KUKA KRL program: EPS_2_25990_SANMH01_A_20251014010954.src

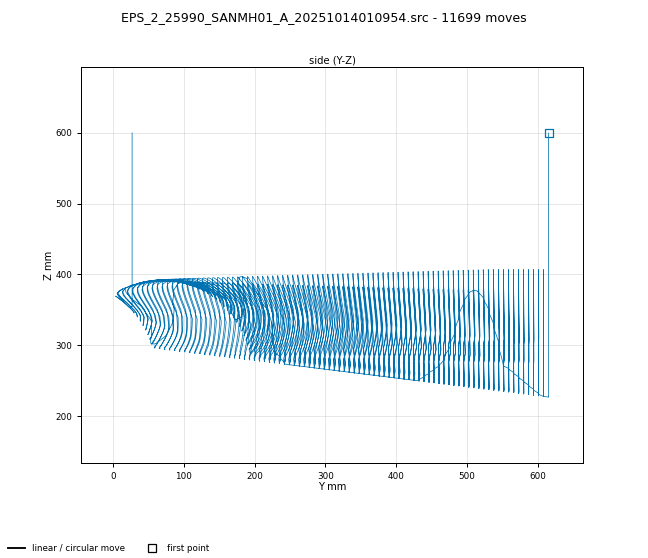
[picture p0: tool path of EPS_2_25990_SANMH01_A_20251014010954.src, 11699 of 11701 moves have a stored position in this frame; points joined in program order, loops and branches not executed]
&ACCESS RVP
&REL 4
&COMMENT QRS 19112012
&PARAM EDITMASK = *
DEF PART()
EXT BAS (BAS_COMMAND :IN,REAL :IN )
INT I
BAS (#INITMOV,0 )

;KUKA QRS Post kuka4.cps  Date:22-06-2017 !

File_ID=2882

QRS_PRE_INIT()

;Init var - Until changes are made in qrs_pre_init
Outlet_Square_prg=0
Inlet_1_Square_prg=0
Inlet_2_Square_prg=0
Inlet_3_Square_prg=0
Inlet_4_Square_prg=0
Inlet_5_Square_prg=0

Outlet_1={X 0.000, Y 531.880, Z 306.500, B 0.000, E1 0.000 }
Inlet_1={X 0.000, Y 534.050, Z 276.500, B 0.000, E1 136.000 }
Outlet_1_type=201
Inlet_1_type=201
;QRS#1=Sidecore dimensions
;QRS#2=200-8" PVC SDR 35
;QRS#3=200-8" PVC SDR 35
;QRS#4=
;QRS#5=
;QRS#6=
;QRS#7=
;QRS#8=
;QRS#9=12-08 PSX
;QRS#10=12-08 PSX
;QRS#11=
;QRS#12=
;QRS#13=
;QRS#14=
;QRS#15=
;QRS#16=1220x127x686 2,25'
;QRS#17=EPS Height
;QRS#18=407
;QRS#19=*
;QRS#20= UPDATED VERSION 22-06-2017
;QRS#21=*
Outlet_Square=0100
Inlet_1_Square=0100
Inlet_2_Square=0
Inlet_3_Square=0
Inlet_4_Square=0
Inlet_5_Square=0
Mill_Square=1
Outlet_Square_Prg=204
Inlet_1_Square_prg=204

QRS_INIT()

$ADVANCE=5

; T1
PTP {E1 173.591,E2 173.591}
PTP {X 0,Y 615.515,A -85,B 0,C 180,E1 173.591,E2 173.591,E3 0,E4 0,E5 0,E6 0}
QRS_SPEED_INIT()
LIN {X 0,Y 615.515,Z 600,A -85,B 0,C 180,E1 173.591,E2 173.591,E3 0,E4 0,E5 0,E6 0} C_VEL
LIN {X 0,Y 615.515,Z 236.872,A -85,B 0,C 180,E1 173.591,E2 173.591} C_VEL
LIN {X 0,Y 615.515,Z 228.698,A -85,B 0,C 180,E1 173.591,E2 173.591} C_VEL
LIN {X 0,Y 615.495,Z 226.698,A -85,B 0,C 180,E1 173.405,E2 173.405} C_VEL
LIN {X 0,Y 615.477,Z 226.7,A -85,B 0,C 180,E1 170.802,E2 170.802} C_VEL
LIN {X 0,Y 615.494,Z 226.697,A -85,B 0,C 180,E1 169.474,E2 169.474} C_VEL
LIN {X 0,Y 615.459,Z 228.778,A -85,B 0,C 180,E1 168.14,E2 168.14} C_VEL
LIN {X 0,Y 615.473,Z 233.515,A -85,B 0,C 180,E1 165.452,E2 165.452} C_VEL
LIN {X 0,Y 615.488,Z 238.387,A -85,B 0,C 180,E1 162.73,E2 162.73} C_VEL
LIN {X 0,Y 615.488,Z 243.54,A -85,B 0,C 180,E1 159.968,E2 159.968} C_VEL
LIN {X 0,Y 615.486,Z 248.916,A -85,B 0,C 180,E1 157.156,E2 157.156} C_VEL
LIN {X 0,Y 615.468,Z 254.224,A -85,B 0,C 180,E1 154.432,E2 154.432} C_VEL
LIN {X 0,Y 615.487,Z 259.957,A -85,B 0,C 180,E1 151.548,E2 151.548} C_VEL
LIN {X 0,Y 615.466,Z 265.253,A -85,B 0,C 180,E1 148.915,E2 148.915} C_VEL
LIN {X 0,Y 615.466,Z 270.245,A -85,B 0,C 180,E1 146.467,E2 146.467} C_VEL
LIN {X 0,Y 615.49,Z 272.215,A -85,B 0,C 180,E1 145.555,E2 145.555} C_VEL
LIN {X 0,Y 615.481,Z 285.466,A -85,B 0,C 180,E1 145.27,E2 145.27} C_VEL
LIN {X 0,Y 615.458,Z 298.826,A -85,B 0,C 180,E1 144.835,E2 144.835} C_VEL
LIN {X 0,Y 615.475,Z 310.215,A -85,B 0,C 180,E1 144.329,E2 144.329} C_VEL
LIN {X 0,Y 615.489,Z 322.006,A -85,B 0,C 180,E1 143.65,E2 143.65} C_VEL
LIN {X 0,Y 615.498,Z 332.274,A -85,B 0,C 180,E1 142.91,E2 142.91} C_VEL
LIN {X 0,Y 615.495,Z 340.609,A -85,B 0,C 180,E1 142.18,E2 142.18} C_VEL
LIN {X 0,Y 615.497,Z 348.841,A -85,B 0,C 180,E1 141.308,E2 141.308} C_VEL
LIN {X 0,Y 615.494,Z 356.847,A -85,B 0,C 180,E1 140.252,E2 140.252} C_VEL
LIN {X 0,Y 615.495,Z 363.456,A -85,B 0,C 180,E1 139.15,E2 139.15} C_VEL
LIN {X 0,Y 615.495,Z 367.798,A -85,B 0,C 180,E1 138.224,E2 138.224} C_VEL
LIN {X 0,Y 615.494,Z 371.164,A -85,B 0,C 180,E1 137.301,E2 137.301} C_VEL
LIN {X 0,Y 615.493,Z 374.47,A -85,B 0,C 180,E1 136.001,E2 136.001} C_VEL
LIN {X 0,Y 615.493,Z 375.946,A -85,B 0,C 180,E1 134.934,E2 134.934} C_VEL
LIN {X 0,Y 615.493,Z 376.384,A -85,B 0,C 180,E1 134,E2 134} C_VEL
LIN {X 0,Y 615.492,Z 375.997,A -85,B 0,C 180,E1 133.05,E2 133.05} C_VEL
LIN {X 0,Y 615.494,Z 374.759,A -85,B 0,C 180,E1 132.083,E2 132.083} C_VEL
LIN {X 0,Y 615.495,Z 372.591,A -85,B 0,C 180,E1 131.097,E2 131.097} C_VEL
LIN {X 0,Y 615.496,Z 369.385,A -85,B 0,C 180,E1 130.092,E2 130.092} C_VEL
LIN {X 0,Y 615.493,Z 364.194,A -85,B 0,C 180,E1 128.903,E2 128.903} C_VEL
LIN {X 0,Y 615.497,Z 357.942,A -85,B 0,C 180,E1 127.82,E2 127.82} C_VEL
LIN {X 0,Y 615.493,Z 350.544,A -85,B 0,C 180,E1 126.81,E2 126.81} C_VEL
LIN {X 0,Y 615.498,Z 341.718,A -85,B 0,C 180,E1 125.837,E2 125.837} C_VEL
LIN {X 0,Y 615.497,Z 332.446,A -85,B 0,C 180,E1 125.013,E2 125.013} C_VEL
LIN {X 0,Y 615.465,Z 320.994,A -85,B 0,C 180,E1 124.193,E2 124.193} C_VEL
LIN {X 0,Y 615.415,Z 310.393,A -85,B 0,C 180,E1 123.588,E2 123.588} C_VEL
LIN {X 0,Y 615.427,Z 298.003,A -85,B 0,C 180,E1 123.044,E2 123.044} C_VEL
LIN {X 0,Y 615.47,Z 285.899,A -85,B 0,C 180,E1 122.652,E2 122.652} C_VEL
LIN {X 0,Y 615.479,Z 272.071,A -85,B 0,C 180,E1 122.332,E2 122.332} C_VEL
LIN {X 0,Y 615.417,Z 266.106,A -85,B 0,C 180,E1 119.409,E2 119.409} C_VEL
LIN {X 0,Y 615.448,Z 261.314,A -85,B 0,C 180,E1 117.041,E2 117.041} C_VEL
LIN {X 0,Y 615.457,Z 255.808,A -85,B 0,C 180,E1 114.273,E2 114.273} C_VEL
LIN {X 0,Y 615.443,Z 251.613,A -85,B 0,C 180,E1 112.138,E2 112.138} C_VEL
LIN {X 0,Y 615.436,Z 247.54,A -85,B 0,C 180,E1 110.034,E2 110.034} C_VEL
LIN {X 0,Y 615.433,Z 243.584,A -85,B 0,C 180,E1 107.958,E2 107.958} C_VEL
LIN {X 0,Y 615.436,Z 239.741,A -85,B 0,C 180,E1 105.906,E2 105.906} C_VEL
LIN {X 0,Y 615.485,Z 234.819,A -85,B 0,C 180,E1 103.201,E2 103.201} C_VEL
LIN {X 0,Y 615.495,Z 230.063,A -85,B 0,C 180,E1 100.526,E2 100.526} C_VEL
LIN {X 0,Y 615.478,Z 226.7,A -85,B 0,C 180,E1 98.536,E2 98.536} C_VEL
LIN {X 0,Y 615.468,Z 226.7,A -85,B 0,C 180,E1 95.899,E2 95.899} C_VEL
LIN {X 0,Y 615.476,Z 226.698,A -85,B 0,C 180,E1 93.273,E2 93.273} C_VEL
LIN {X 0,Y 615.489,Z 226.697,A -85,B 0,C 180,E1 90.654,E2 90.654} C_VEL
LIN {X 0,Y 615.495,Z 226.7,A -85,B 0,C 180,E1 88.037,E2 88.037} C_VEL
LIN {X 0,Y 615.495,Z 226.698,A -85,B 0,C 180,E1 85.415,E2 85.415} C_VEL
LIN {X 0,Y 615.475,Z 226.699,A -85,B 0,C 180,E1 82.784,E2 82.784} C_VEL
LIN {X 0,Y 615.464,Z 226.701,A -85,B 0,C 180,E1 80.138,E2 80.138} C_VEL
LIN {X 0,Y 615.478,Z 226.699,A -85,B 0,C 180,E1 77.47,E2 77.47} C_VEL
LIN {X 0,Y 615.492,Z 226.702,A -85,B 0,C 180,E1 74.774,E2 74.774} C_VEL
LIN {X 0,Y 615.475,Z 226.699,A -85,B 0,C 180,E1 72.043,E2 72.043} C_VEL
LIN {X 0,Y 615.492,Z 226.694,A -85,B 0,C 180,E1 69.27,E2 69.27} C_VEL
LIN {X 0,Y 615.484,Z 226.702,A -85,B 0,C 180,E1 66.444,E2 66.444} C_VEL
LIN {X 0,Y 615.493,Z 226.695,A -85,B 0,C 180,E1 63.557,E2 63.557} C_VEL
LIN {X 0,Y 615.482,Z 226.7,A -85,B 0,C 180,E1 60.594,E2 60.594} C_VEL
LIN {X 0,Y 615.473,Z 226.7,A -85,B 0,C 180,E1 58.314,E2 58.314} C_VEL
LIN {X 0,Y 615.469,Z 226.7,A -85,B 0,C 180,E1 55.977,E2 55.977} C_VEL
LIN {X 0,Y 615.491,Z 226.695,A -85,B 0,C 180,E1 53.576,E2 53.576} C_VEL
LIN {X 0,Y 615.49,Z 226.699,A -85,B 0,C 180,E1 50.936,E2 50.936} C_VEL
LIN {X 0,Y 615.484,Z 226.7,A -85,B 0,C 180,E1 48.527,E2 48.527} C_VEL
LIN {X 0,Y 615.499,Z 226.698,A -85,B 0,C 180,E1 45.852,E2 45.852} C_VEL
LIN {X 0,Y 615.465,Z 226.7,A -85,B 0,C 180,E1 43.046,E2 43.046} C_VEL
LIN {X 0,Y 615.467,Z 226.7,A -85,B 0,C 180,E1 40.607,E2 40.607} C_VEL
LIN {X 0,Y 615.484,Z 226.697,A -85,B 0,C 180,E1 38.013,E2 38.013} C_VEL
LIN {X 0,Y 615.487,Z 226.696,A -85,B 0,C 180,E1 35.615,E2 35.615} C_VEL
LIN {X 0,Y 615.47,Z 226.7,A -85,B 0,C 180,E1 33.236,E2 33.236} C_VEL
LIN {X 0,Y 615.467,Z 226.7,A -85,B 0,C 180,E1 30.92,E2 30.92} C_VEL
LIN {X 0,Y 615.472,Z 226.699,A -85,B 0,C 180,E1 28.449,E2 28.449} C_VEL
LIN {X 0,Y 615.498,Z 226.7,A -85,B 0,C 180,E1 25.573,E2 25.573} C_VEL
LIN {X 0,Y 615.477,Z 226.699,A -85,B 0,C 180,E1 22.844,E2 22.844} C_VEL
LIN {X 0,Y 615.493,Z 226.694,A -85,B 0,C 180,E1 20.032,E2 20.032} C_VEL
LIN {X 0,Y 615.488,Z 226.701,A -85,B 0,C 180,E1 17.269,E2 17.269} C_VEL
LIN {X 0,Y 615.494,Z 226.697,A -85,B 0,C 180,E1 14.548,E2 14.548} C_VEL
LIN {X 0,Y 615.472,Z 226.699,A -85,B 0,C 180,E1 11.86,E2 11.86} C_VEL
LIN {X 0,Y 615.469,Z 226.7,A -85,B 0,C 180,E1 9.198,E2 9.198} C_VEL
LIN {X 0,Y 615.485,Z 226.7,A -85,B 0,C 180,E1 6.556,E2 6.556} C_VEL
LIN {X 0,Y 615.487,Z 226.702,A -85,B 0,C 180,E1 3.928,E2 3.928} C_VEL
LIN {X 0,Y 615.48,Z 226.699,A -85,B 0,C 180,E1 1.308,E2 1.308} C_VEL
LIN {X 0,Y 615.493,Z 226.694,A -85,B 0,C 180,E1 -1.309,E2 -1.309} C_VEL
LIN {X 0,Y 615.477,Z 226.698,A -85,B 0,C 180,E1 -3.929,E2 -3.929} C_VEL
LIN {X 0,Y 615.477,Z 226.7,A -85,B 0,C 180,E1 -6.578,E2 -6.578} C_VEL
LIN {X 0,Y 615.496,Z 226.7,A -85,B 0,C 180,E1 -9.199,E2 -9.199} C_VEL
LIN {X 0,Y 615.479,Z 226.7,A -85,B 0,C 180,E1 -11.862,E2 -11.862} C_VEL
LIN {X 0,Y 615.467,Z 226.7,A -85,B 0,C 180,E1 -14.55,E2 -14.55} C_VEL
LIN {X 0,Y 615.496,Z 226.695,A -85,B 0,C 180,E1 -17.271,E2 -17.271} C_VEL
LIN {X 0,Y 615.489,Z 226.702,A -85,B 0,C 180,E1 -20.033,E2 -20.033} C_VEL
LIN {X 0,Y 615.489,Z 226.696,A -85,B 0,C 180,E1 -22.845,E2 -22.845} C_VEL
LIN {X 0,Y 615.477,Z 226.699,A -85,B 0,C 180,E1 -25.717,E2 -25.717} C_VEL
LIN {X 0,Y 615.499,Z 226.7,A -85,B 0,C 180,E1 -28.454,E2 -28.454} C_VEL
LIN {X 0,Y 615.486,Z 226.698,A -85,B 0,C 180,E1 -31.087,E2 -31.087} C_VEL
LIN {X 0,Y 615.475,Z 226.7,A -85,B 0,C 180,E1 -33.534,E2 -33.534} C_VEL
LIN {X 0,Y 615.481,Z 226.7,A -85,B 0,C 180,E1 -35.834,E2 -35.834} C_VEL
LIN {X 0,Y 615.488,Z 226.702,A -85,B 0,C 180,E1 -38.069,E2 -38.069} C_VEL
LIN {X 0,Y 615.486,Z 226.696,A -85,B 0,C 180,E1 -41.095,E2 -41.095} C_VEL
LIN {X 0,Y 615.493,Z 226.699,A -85,B 0,C 180,E1 -44.15,E2 -44.15} C_VEL
LIN {X 0,Y 615.485,Z 226.696,A -85,B 0,C 180,E1 -46.953,E2 -46.953} C_VEL
LIN {X 0,Y 615.467,Z 226.7,A -85,B 0,C 180,E1 -49.393,E2 -49.393} C_VEL
LIN {X 0,Y 615.469,Z 226.7,A -85,B 0,C 180,E1 -51.991,E2 -51.991} C_VEL
LIN {X 0,Y 615.491,Z 226.813,A -85,B 0,C 180,E1 -54.586,E2 -54.586} C_VEL
LIN {X 0,Y 615.479,Z 233.99,A -85,B 0,C 180,E1 -57.154,E2 -57.154} C_VEL
LIN {X 0,Y 615.46,Z 241.78,A -85,B 0,C 180,E1 -59.839,E2 -59.839} C_VEL
LIN {X 0,Y 615.492,Z 249.544,A -85,B 0,C 180,E1 -62.455,E2 -62.455} C_VEL
LIN {X 0,Y 615.442,Z 257.313,A -85,B 0,C 180,E1 -65.007,E2 -65.007} C_VEL
LIN {X 0,Y 615.47,Z 265.535,A -85,B 0,C 180,E1 -67.659,E2 -67.659} C_VEL
LIN {X 0,Y 615.487,Z 273.927,A -85,B 0,C 180,E1 -70.315,E2 -70.315} C_VEL
LIN {X 0,Y 615.484,Z 282.785,A -85,B 0,C 180,E1 -73.072,E2 -73.072} C_VEL
LIN {X 0,Y 615.469,Z 291.547,A -85,B 0,C 180,E1 -75.76,E2 -75.76} C_VEL
LIN {X 0,Y 615.496,Z 300.138,A -85,B 0,C 180,E1 -78.369,E2 -78.369} C_VEL
LIN {X 0,Y 615.497,Z 313.826,A -85,B 0,C 180,E1 -78.64,E2 -78.64} C_VEL
LIN {X 0,Y 615.455,Z 326.951,A -85,B 0,C 180,E1 -79.05,E2 -79.05} C_VEL
LIN {X 0,Y 615.447,Z 338.775,A -85,B 0,C 180,E1 -79.556,E2 -79.556} C_VEL
LIN {X 0,Y 615.497,Z 349.388,A -85,B 0,C 180,E1 -80.138,E2 -80.138} C_VEL
LIN {X 0,Y 615.498,Z 360.233,A -85,B 0,C 180,E1 -80.884,E2 -80.884} C_VEL
LIN {X 0,Y 615.497,Z 370.812,A -85,B 0,C 180,E1 -81.794,E2 -81.794} C_VEL
LIN {X 0,Y 615.498,Z 378.606,A -85,B 0,C 180,E1 -82.62,E2 -82.62} C_VEL
LIN {X 0,Y 615.496,Z 386.203,A -85,B 0,C 180,E1 -83.608,E2 -83.608} C_VEL
LIN {X 0,Y 615.498,Z 393.204,A -85,B 0,C 180,E1 -84.759,E2 -84.759} C_VEL
LIN {X 0,Y 615.494,Z 397.851,A -85,B 0,C 180,E1 -85.744,E2 -85.744} C_VEL
LIN {X 0,Y 615.494,Z 401.399,A -85,B 0,C 180,E1 -86.727,E2 -86.727} C_VEL
LIN {X 0,Y 615.497,Z 403.233,A -85,B 0,C 180,E1 -87.382,E2 -87.382} C_VEL
LIN {X 0,Y 615.5,Z 404.607,A -85,B 0,C 180,E1 -88.037,E2 -88.037} C_VEL
LIN {X 0,Y 615.496,Z 406.173,A -85,B 0,C 180,E1 -89.346,E2 -89.346} C_VEL
LIN {X 0,Y 615.494,Z 406.389,A -85,B 0,C 180,E1 -90,E2 -90} C_VEL
LIN {X 0,Y 615.495,Z 405.58,A -85,B 0,C 180,E1 -91.308,E2 -91.308} C_VEL
LIN {X 0,Y 615.5,Z 404.608,A -85,B 0,C 180,E1 -91.963,E2 -91.963} C_VEL
LIN {X 0,Y 615.497,Z 403.233,A -85,B 0,C 180,E1 -92.618,E2 -92.618} C_VEL
LIN {X 0,Y 615.496,Z 400.35,A -85,B 0,C 180,E1 -93.6,E2 -93.6} C_VEL
LIN {X 0,Y 615.498,Z 396.442,A -85,B 0,C 180,E1 -94.584,E2 -94.584} C_VEL
LIN {X 0,Y 615.499,Z 391.406,A -85,B 0,C 180,E1 -95.569,E2 -95.569} C_VEL
LIN {X 0,Y 615.497,Z 384.871,A -85,B 0,C 180,E1 -96.583,E2 -96.583} C_VEL
LIN {X 0,Y 615.497,Z 377.135,A -85,B 0,C 180,E1 -97.545,E2 -97.545} C_VEL
LIN {X 0,Y 615.498,Z 369.048,A -85,B 0,C 180,E1 -98.371,E2 -98.371} C_VEL
LIN {X 0,Y 615.499,Z 359.171,A -85,B 0,C 180,E1 -99.198,E2 -99.198} C_VEL
LIN {X 0,Y 615.486,Z 347.987,A -85,B 0,C 180,E1 -99.945,E2 -99.945} C_VEL
LIN {X 0,Y 615.445,Z 337.036,A -85,B 0,C 180,E1 -100.527,E2 -100.527} C_VEL
LIN {X 0,Y 615.461,Z 324.766,A -85,B 0,C 180,E1 -101.031,E2 -101.031} C_VEL
LIN {X 0,Y 615.498,Z 312.077,A -85,B 0,C 180,E1 -101.401,E2 -101.401} C_VEL
LIN {X 0,Y 615.496,Z 300.139,A -85,B 0,C 180,E1 -101.631,E2 -101.631} C_VEL
LIN {X 0,Y 615.469,Z 291.548,A -85,B 0,C 180,E1 -104.24,E2 -104.24} C_VEL
LIN {X 0,Y 615.484,Z 282.786,A -85,B 0,C 180,E1 -106.928,E2 -106.928} C_VEL
LIN {X 0,Y 615.487,Z 273.928,A -85,B 0,C 180,E1 -109.684,E2 -109.684} C_VEL
LIN {X 0,Y 615.474,Z 265.532,A -85,B 0,C 180,E1 -112.342,E2 -112.342} C_VEL
LIN {X 0,Y 615.442,Z 257.313,A -85,B 0,C 180,E1 -114.993,E2 -114.993} C_VEL
LIN {X 0,Y 615.492,Z 249.545,A -85,B 0,C 180,E1 -117.545,E2 -117.545} C_VEL
LIN {X 0,Y 615.46,Z 241.779,A -85,B 0,C 180,E1 -120.161,E2 -120.161} C_VEL
LIN {X 0,Y 615.478,Z 233.974,A -85,B 0,C 180,E1 -122.846,E2 -122.846} C_VEL
LIN {X 0,Y 615.492,Z 226.697,A -85,B 0,C 180,E1 -125.514,E2 -125.514} C_VEL
LIN {X 0,Y 615.488,Z 226.699,A -85,B 0,C 180,E1 -128.068,E2 -128.068} C_VEL
LIN {X 0,Y 615.48,Z 226.7,A -85,B 0,C 180,E1 -130.606,E2 -130.606} C_VEL
LIN {X 0,Y 615.497,Z 226.698,A -85,B 0,C 180,E1 -133.243,E2 -133.243} C_VEL
LIN {X 0,Y 615.476,Z 226.7,A -85,B 0,C 180,E1 -136.002,E2 -136.002} C_VEL
LIN {X 0,Y 615.49,Z 226.697,A -85,B 0,C 180,E1 -138.904,E2 -138.904} C_VEL
LIN {X 0,Y 615.495,Z 226.696,A -85,B 0,C 180,E1 -141.096,E2 -141.096} C_VEL
LIN {X 0,Y 615.491,Z 226.701,A -85,B 0,C 180,E1 -143.575,E2 -143.575} C_VEL
LIN {X 0,Y 615.481,Z 226.7,A -85,B 0,C 180,E1 -145.977,E2 -145.977} C_VEL
LIN {X 0,Y 615.473,Z 226.701,A -85,B 0,C 180,E1 -148.313,E2 -148.313} C_VEL
LIN {X 0,Y 615.478,Z 226.701,A -85,B 0,C 180,E1 -150.593,E2 -150.593} C_VEL
LIN {X 0,Y 615.498,Z 226.699,A -85,B 0,C 180,E1 -152.951,E2 -152.951} C_VEL
LIN {X 0,Y 615.494,Z 226.701,A -85,B 0,C 180,E1 -155.988,E2 -155.988} C_VEL
LIN {X 0,Y 615.484,Z 226.698,A -85,B 0,C 180,E1 -158.567,E2 -158.567} C_VEL
LIN {X 0,Y 615.48,Z 226.7,A -85,B 0,C 180,E1 -161.394,E2 -161.394} C_VEL
LIN {X 0,Y 615.486,Z 226.701,A -85,B 0,C 180,E1 -164.094,E2 -164.094} C_VEL
LIN {X 0,Y 615.497,Z 226.695,A -85,B 0,C 180,E1 -166.798,E2 -166.798} C_VEL
LIN {X 0,Y 615.484,Z 226.701,A -85,B 0,C 180,E1 -169.472,E2 -169.472} C_VEL
LIN {X 0,Y 615.481,Z 226.7,A -85,B 0,C 180,E1 -172.124,E2 -172.124} C_VEL
LIN {X 0,Y 615.489,Z 226.698,A -85,B 0,C 180,E1 -174.758,E2 -174.758} C_VEL
LIN {X 0,Y 615.489,Z 226.7,A -85,B 0,C 180,E1 -177.381,E2 -177.381} C_VEL
LIN {X 0,Y 615.478,Z 226.7,A -85,B 0,C 180,E1 -179.999,E2 -179.999} C_VEL
LIN {X 0,Y 615.495,Z 226.7,A -85,B 0,C 180,E1 -182.617,E2 -182.617} C_VEL
LIN {X 0,Y 615.474,Z 226.7,A -85,B 0,C 180,E1 -185.24,E2 -185.24} C_VEL
LIN {X 0,Y 615.495,Z 226.698,A -85,B 0,C 180,E1 -186.595,E2 -186.595} C_VEL
LIN {X 0,Y 614.805,Z 226.845,A -85,B 0,C 180,E1 -187.141,E2 -187.141} C_VEL
LIN {X 0,Y 611.958,Z 227.26,A -85,B 0,C 180,E1 -188.027,E2 -188.027} C_VEL
LIN {X 0,Y 609.568,Z 227.568,A -85,B 0,C 180,E1 -188.739,E2 -188.739} C_VEL
LIN {X 0,Y 608.541,Z 227.685,A -85,B 0,C 180,E1 -189.289,E2 -189.289} C_VEL
LIN {X 0,Y 608.457,Z 227.694,A -85,B 0,C 180,E1 -189.475,E2 -189.475} C_VEL
LIN {X 0,Y 608.443,Z 227.698,A -85,B 0,C 180,E1 -190.649,E2 -190.649} C_VEL
LIN {X 0,Y 608.431,Z 232.361,A -85,B 0,C 180,E1 -193.356,E2 -193.356} C_VEL
LIN {X 0,Y 608.445,Z 237.188,A -85,B 0,C 180,E1 -196.093,E2 -196.093} C_VEL
LIN {X 0,Y 608.448,Z 242.225,A -85,B 0,C 180,E1 -198.869,E2 -198.869} C_VEL
LIN {X 0,Y 608.438,Z 247.537,A -85,B 0,C 180,E1 -201.692,E2 -201.692} C_VEL
LIN {X 0,Y 608.424,Z 253.079,A -85,B 0,C 180,E1 -204.571,E2 -204.571} C_VEL
LIN {X 0,Y 608.415,Z 258.231,A -85,B 0,C 180,E1 -207.198,E2 -207.198} C_VEL
LIN {X 0,Y 608.448,Z 263.754,A -85,B 0,C 180,E1 -209.97,E2 -209.97} C_VEL
LIN {X 0,Y 608.414,Z 269.639,A -85,B 0,C 180,E1 -212.881,E2 -212.881} C_VEL
LIN {X 0,Y 608.442,Z 272.542,A -85,B 0,C 180,E1 -214.305,E2 -214.305} C_VEL
LIN {X 0,Y 608.52,Z 287.737,A -85,B 0,C 180,E1 -214.659,E2 -214.659} C_VEL
LIN {X 0,Y 608.501,Z 299.429,A -85,B 0,C 180,E1 -215.057,E2 -215.057} C_VEL
LIN {X 0,Y 608.478,Z 310.914,A -85,B 0,C 180,E1 -215.579,E2 -215.579} C_VEL
LIN {X 0,Y 608.496,Z 323.052,A -85,B 0,C 180,E1 -216.292,E2 -216.292} C_VEL
LIN {X 0,Y 608.485,Z 333.177,A -85,B 0,C 180,E1 -217.037,E2 -217.037} C_VEL
LIN {X 0,Y 608.468,Z 342.371,A -85,B 0,C 180,E1 -217.868,E2 -217.868} C_VEL
LIN {X 0,Y 608.444,Z 350.491,A -85,B 0,C 180,E1 -218.765,E2 -218.765} C_VEL
LIN {X 0,Y 608.437,Z 357.135,A -85,B 0,C 180,E1 -219.655,E2 -219.655} C_VEL
LIN {X 0,Y 608.435,Z 363.654,A -85,B 0,C 180,E1 -220.738,E2 -220.738} C_VEL
LIN {X 0,Y 608.449,Z 368.088,A -85,B 0,C 180,E1 -221.673,E2 -221.673} C_VEL
LIN {X 0,Y 608.438,Z 370.653,A -85,B 0,C 180,E1 -222.333,E2 -222.333} C_VEL
LIN {X 0,Y 608.431,Z 373.569,A -85,B 0,C 180,E1 -223.306,E2 -223.306} C_VEL
LIN {X 0,Y 608.418,Z 375.537,A -85,B 0,C 180,E1 -224.261,E2 -224.261} C_VEL
LIN {X 0,Y 608.415,Z 376.656,A -85,B 0,C 180,E1 -225.202,E2 -225.202} C_VEL
LIN {X 0,Y 608.426,Z 376.987,A -85,B 0,C 180,E1 -226.128,E2 -226.128} C_VEL
LIN {X 0,Y 608.431,Z 376.549,A -85,B 0,C 180,E1 -227.039,E2 -227.039} C_VEL
LIN {X 0,Y 608.422,Z 375.358,A -85,B 0,C 180,E1 -227.936,E2 -227.936} C_VEL
LIN {X 0,Y 608.431,Z 373.465,A -85,B 0,C 180,E1 -228.823,E2 -228.823} C_VEL
LIN {X 0,Y 608.438,Z 370.866,A -85,B 0,C 180,E1 -229.697,E2 -229.697} C_VEL
LIN {X 0,Y 608.45,Z 366.862,A -85,B 0,C 180,E1 -230.703,E2 -230.703} C_VEL
LIN {X 0,Y 608.434,Z 361.387,A -85,B 0,C 180,E1 -231.762,E2 -231.762} C_VEL
LIN {X 0,Y 608.443,Z 354.246,A -85,B 0,C 180,E1 -232.843,E2 -232.843} C_VEL
LIN {X 0,Y 608.459,Z 347.242,A -85,B 0,C 180,E1 -233.705,E2 -233.705} C_VEL
LIN {X 0,Y 608.476,Z 338.162,A -85,B 0,C 180,E1 -234.624,E2 -234.624} C_VEL
LIN {X 0,Y 608.477,Z 328.441,A -85,B 0,C 180,E1 -235.421,E2 -235.421} C_VEL
LIN {X 0,Y 608.437,Z 316.606,A -85,B 0,C 180,E1 -236.2,E2 -236.2} C_VEL
LIN {X 0,Y 608.429,Z 305.532,A -85,B 0,C 180,E1 -236.774,E2 -236.774} C_VEL
LIN {X 0,Y 608.488,Z 294.204,A -85,B 0,C 180,E1 -237.228,E2 -237.228} C_VEL
LIN {X 0,Y 608.533,Z 281.365,A -85,B 0,C 180,E1 -237.597,E2 -237.597} C_VEL
LIN {X 0,Y 608.398,Z 272.531,A -85,B 0,C 180,E1 -237.792,E2 -237.792} C_VEL
LIN {X 0,Y 608.373,Z 267.597,A -85,B 0,C 180,E1 -240.216,E2 -240.216} C_VEL
LIN {X 0,Y 608.387,Z 262.38,A -85,B 0,C 180,E1 -242.807,E2 -242.807} C_VEL
LIN {X 0,Y 608.397,Z 257.176,A -85,B 0,C 180,E1 -245.427,E2 -245.427} C_VEL
LIN {X 0,Y 608.418,Z 252.935,A -85,B 0,C 180,E1 -247.593,E2 -247.593} C_VEL
LIN {X 0,Y 608.399,Z 248.827,A -85,B 0,C 180,E1 -249.724,E2 -249.724} C_VEL
LIN {X 0,Y 608.42,Z 243.53,A -85,B 0,C 180,E1 -252.523,E2 -252.523} C_VEL
LIN {X 0,Y 608.433,Z 238.464,A -85,B 0,C 180,E1 -255.279,E2 -255.279} C_VEL
LIN {X 0,Y 608.461,Z 233.611,A -85,B 0,C 180,E1 -258.001,E2 -258.001} C_VEL
LIN {X 0,Y 608.42,Z 228.894,A -85,B 0,C 180,E1 -260.694,E2 -260.694} C_VEL
LIN {X 0,Y 608.446,Z 227.736,A -85,B 0,C 180,E1 -261.364,E2 -261.364} C_VEL
LIN {X 0,Y 608.445,Z 227.696,A -85,B 0,C 180,E1 -264.033,E2 -264.033} C_VEL
LIN {X 0,Y 608.469,Z 227.692,A -85,B 0,C 180,E1 -266.689,E2 -266.689} C_VEL
LIN {X 0,Y 608.482,Z 227.692,A -85,B 0,C 180,E1 -269.338,E2 -269.338} C_VEL
LIN {X 0,Y 608.464,Z 227.697,A -85,B 0,C 180,E1 -271.986,E2 -271.986} C_VEL
LIN {X 0,Y 608.462,Z 227.695,A -85,B 0,C 180,E1 -274.638,E2 -274.638} C_VEL
LIN {X 0,Y 608.455,Z 227.694,A -85,B 0,C 180,E1 -277.299,E2 -277.299} C_VEL
LIN {X 0,Y 608.44,Z 227.696,A -85,B 0,C 180,E1 -279.977,E2 -279.977} C_VEL
LIN {X 0,Y 608.466,Z 227.695,A -85,B 0,C 180,E1 -282.677,E2 -282.677} C_VEL
LIN {X 0,Y 608.469,Z 227.694,A -85,B 0,C 180,E1 -285.406,E2 -285.406} C_VEL
LIN {X 0,Y 608.442,Z 227.696,A -85,B 0,C 180,E1 -288.172,E2 -288.172} C_VEL
LIN {X 0,Y 608.455,Z 227.696,A -85,B 0,C 180,E1 -290.981,E2 -290.981} C_VEL
LIN {X 0,Y 608.447,Z 227.695,A -85,B 0,C 180,E1 -293.124,E2 -293.124} C_VEL
LIN {X 0,Y 608.455,Z 227.695,A -85,B 0,C 180,E1 -295.72,E2 -295.72} C_VEL
LIN {X 0,Y 608.452,Z 227.697,A -85,B 0,C 180,E1 -298.266,E2 -298.266} C_VEL
LIN {X 0,Y 608.47,Z 227.693,A -85,B 0,C 180,E1 -300.544,E2 -300.544} C_VEL
LIN {X 0,Y 608.458,Z 227.694,A -85,B 0,C 180,E1 -302.879,E2 -302.879} C_VEL
LIN {X 0,Y 608.441,Z 227.696,A -85,B 0,C 180,E1 -305.277,E2 -305.277} C_VEL
LIN {X 0,Y 608.469,Z 227.694,A -85,B 0,C 180,E1 -308.242,E2 -308.242} C_VEL
LIN {X 0,Y 608.47,Z 227.695,A -85,B 0,C 180,E1 -310.333,E2 -310.333} C_VEL
LIN {X 0,Y 608.445,Z 227.698,A -85,B 0,C 180,E1 -312.96,E2 -312.96} C_VEL
LIN {X 0,Y 608.447,Z 227.695,A -85,B 0,C 180,E1 -315.736,E2 -315.736} C_VEL
LIN {X 0,Y 608.463,Z 227.695,A -85,B 0,C 180,E1 -318.657,E2 -318.657} C_VEL
LIN {X 0,Y 608.466,Z 227.695,A -85,B 0,C 180,E1 -321.413,E2 -321.413} C_VEL
LIN {X 0,Y 608.472,Z 227.693,A -85,B 0,C 180,E1 -323.95,E2 -323.95} C_VEL
LIN {X 0,Y 608.454,Z 227.695,A -85,B 0,C 180,E1 -326.33,E2 -326.33} C_VEL
LIN {X 0,Y 608.465,Z 227.694,A -85,B 0,C 180,E1 -328.728,E2 -328.728} C_VEL
LIN {X 0,Y 608.459,Z 227.694,A -85,B 0,C 180,E1 -331.381,E2 -331.381} C_VEL
LIN {X 0,Y 608.477,Z 227.694,A -85,B 0,C 180,E1 -334.276,E2 -334.276} C_VEL
LIN {X 0,Y 608.443,Z 227.699,A -85,B 0,C 180,E1 -336.877,E2 -336.877} C_VEL
LIN {X 0,Y 608.466,Z 227.693,A -85,B 0,C 180,E1 -339.727,E2 -339.727} C_VEL
LIN {X 0,Y 608.451,Z 227.696,A -85,B 0,C 180,E1 -342.524,E2 -342.524} C_VEL
LIN {X 0,Y 608.474,Z 227.695,A -85,B 0,C 180,E1 -345.28,E2 -345.28} C_VEL
LIN {X 0,Y 608.449,Z 227.695,A -85,B 0,C 180,E1 -348.001,E2 -348.001} C_VEL
LIN {X 0,Y 608.457,Z 227.694,A -85,B 0,C 180,E1 -350.695,E2 -350.695} C_VEL
LIN {X 0,Y 608.468,Z 227.694,A -85,B 0,C 180,E1 -353.368,E2 -353.368} C_VEL
LIN {X 0,Y 608.456,Z 227.698,A -85,B 0,C 180,E1 -356.027,E2 -356.027} C_VEL
LIN {X 0,Y 608.463,Z 227.694,A -85,B 0,C 180,E1 -358.677,E2 -358.677} C_VEL
LIN {X 0,Y 608.475,Z 227.692,A -85,B 0,C 180,E1 -361.324,E2 -361.324} C_VEL
LIN {X 0,Y 608.447,Z 227.695,A -85,B 0,C 180,E1 -363.975,E2 -363.975} C_VEL
LIN {X 0,Y 608.47,Z 227.694,A -85,B 0,C 180,E1 -366.633,E2 -366.633} C_VEL
LIN {X 0,Y 608.475,Z 227.695,A -85,B 0,C 180,E1 -369.306,E2 -369.306} C_VEL
LIN {X 0,Y 608.454,Z 227.695,A -85,B 0,C 180,E1 -372.001,E2 -372.001} C_VEL
LIN {X 0,Y 608.463,Z 227.693,A -85,B 0,C 180,E1 -374.721,E2 -374.721} C_VEL
LIN {X 0,Y 608.455,Z 227.696,A -85,B 0,C 180,E1 -377.477,E2 -377.477} C_VEL
LIN {X 0,Y 608.457,Z 227.695,A -85,B 0,C 180,E1 -380.275,E2 -380.275} C_VEL
LIN {X 0,Y 608.453,Z 227.694,A -85,B 0,C 180,E1 -383.125,E2 -383.125} C_VEL
LIN {X 0,Y 608.436,Z 227.7,A -85,B 0,C 180,E1 -386.037,E2 -386.037} C_VEL
LIN {X 0,Y 608.48,Z 227.693,A -85,B 0,C 180,E1 -388.623,E2 -388.623} C_VEL
LIN {X 0,Y 608.473,Z 227.692,A -85,B 0,C 180,E1 -391.317,E2 -391.317} C_VEL
LIN {X 0,Y 608.441,Z 227.696,A -85,B 0,C 180,E1 -393.732,E2 -393.732} C_VEL
LIN {X 0,Y 608.441,Z 227.696,A -85,B 0,C 180,E1 -396.093,E2 -396.093} C_VEL
LIN {X 0,Y 608.474,Z 227.692,A -85,B 0,C 180,E1 -398.588,E2 -398.588} C_VEL
LIN {X 0,Y 608.464,Z 227.694,A -85,B 0,C 180,E1 -401.343,E2 -401.343} C_VEL
LIN {X 0,Y 608.462,Z 227.695,A -85,B 0,C 180,E1 -404.265,E2 -404.265} C_VEL
LIN {X 0,Y 608.453,Z 227.694,A -85,B 0,C 180,E1 -407.041,E2 -407.041} C_VEL
LIN {X 0,Y 608.452,Z 227.695,A -85,B 0,C 180,E1 -409.697,E2 -409.697} C_VEL
LIN {X 0,Y 608.459,Z 227.696,A -85,B 0,C 180,E1 -412.254,E2 -412.254} C_VEL
LIN {X 0,Y 608.479,Z 227.814,A -85,B 0,C 180,E1 -414.472,E2 -414.472} C_VEL
LIN {X 0,Y 608.489,Z 235.135,A -85,B 0,C 180,E1 -417.123,E2 -417.123} C_VEL
LIN {X 0,Y 608.475,Z 241.816,A -85,B 0,C 180,E1 -419.456,E2 -419.456} C_VEL
LIN {X 0,Y 608.439,Z 249.64,A -85,B 0,C 180,E1 -422.108,E2 -422.108} C_VEL
LIN {X 0,Y 608.437,Z 257.432,A -85,B 0,C 180,E1 -424.699,E2 -424.699} C_VEL
LIN {X 0,Y 608.429,Z 265.224,A -85,B 0,C 180,E1 -427.235,E2 -427.235} C_VEL
LIN {X 0,Y 608.456,Z 274.127,A -85,B 0,C 180,E1 -430.078,E2 -430.078} C_VEL
LIN {X 0,Y 608.442,Z 283.031,A -85,B 0,C 180,E1 -432.87,E2 -432.87} C_VEL
LIN {X 0,Y 608.441,Z 290.823,A -85,B 0,C 180,E1 -435.279,E2 -435.279} C_VEL
LIN {X 0,Y 608.453,Z 300.283,A -85,B 0,C 180,E1 -438.169,E2 -438.169} C_VEL
LIN {X 0,Y 608.438,Z 300.492,A -85,B 0,C 180,E1 -438.232,E2 -438.232} C_VEL
LIN {X 0,Y 608.545,Z 314.701,A -85,B 0,C 180,E1 -438.53,E2 -438.53} C_VEL
LIN {X 0,Y 608.497,Z 327.786,A -85,B 0,C 180,E1 -438.95,E2 -438.95} C_VEL
LIN {X 0,Y 608.474,Z 338.924,A -85,B 0,C 180,E1 -439.435,E2 -439.435} C_VEL
LIN {X 0,Y 608.486,Z 349.58,A -85,B 0,C 180,E1 -440.023,E2 -440.023} C_VEL
LIN {X 0,Y 608.483,Z 360.475,A -85,B 0,C 180,E1 -440.778,E2 -440.778} C_VEL
LIN {X 0,Y 608.475,Z 371.112,A -85,B 0,C 180,E1 -441.699,E2 -441.699} C_VEL
LIN {X 0,Y 608.471,Z 378.961,A -85,B 0,C 180,E1 -442.534,E2 -442.534} C_VEL
LIN {X 0,Y 608.461,Z 386.287,A -85,B 0,C 180,E1 -443.485,E2 -443.485} C_VEL
LIN {X 0,Y 608.451,Z 391.866,A -85,B 0,C 180,E1 -444.366,E2 -444.366} C_VEL
LIN {X 0,Y 608.432,Z 396.95,A -85,B 0,C 180,E1 -445.362,E2 -445.362} C_VEL
LIN {X 0,Y 608.449,Z 400.896,A -85,B 0,C 180,E1 -446.358,E2 -446.358} C_VEL
LIN {X 0,Y 608.425,Z 403.809,A -85,B 0,C 180,E1 -447.352,E2 -447.352} C_VEL
LIN {X 0,Y 608.445,Z 405.201,A -85,B 0,C 180,E1 -448.014,E2 -448.014} C_VEL
LIN {X 0,Y 608.438,Z 406.783,A -85,B 0,C 180,E1 -449.338,E2 -449.338} C_VEL
LIN {X 0,Y 608.434,Z 407,A -85,B 0,C 180,E1 -450,E2 -450} C_VEL
LIN {X 0,Y 608.448,Z 406.184,A -85,B 0,C 180,E1 -451.324,E2 -451.324} C_VEL
LIN {X 0,Y 608.445,Z 405.202,A -85,B 0,C 180,E1 -451.986,E2 -451.986} C_VEL
LIN {X 0,Y 608.425,Z 403.81,A -85,B 0,C 180,E1 -452.648,E2 -452.648} C_VEL
LIN {X 0,Y 608.449,Z 400.897,A -85,B 0,C 180,E1 -453.642,E2 -453.642} C_VEL
LIN {X 0,Y 608.432,Z 396.951,A -85,B 0,C 180,E1 -454.638,E2 -454.638} C_VEL
LIN {X 0,Y 608.438,Z 390.878,A -85,B 0,C 180,E1 -455.801,E2 -455.801} C_VEL
LIN {X 0,Y 608.462,Z 384.237,A -85,B 0,C 180,E1 -456.799,E2 -456.799} C_VEL
LIN {X 0,Y 608.456,Z 375.991,A -85,B 0,C 180,E1 -457.8,E2 -457.8} C_VEL
LIN {X 0,Y 608.472,Z 367.539,A -85,B 0,C 180,E1 -458.636,E2 -458.636} C_VEL
LIN {X 0,Y 608.481,Z 357.095,A -85,B 0,C 180,E1 -459.473,E2 -459.473} C_VEL
LIN {X 0,Y 608.494,Z 346.761,A -85,B 0,C 180,E1 -460.144,E2 -460.144} C_VEL
LIN {X 0,Y 608.469,Z 335.846,A -85,B 0,C 180,E1 -460.714,E2 -460.714} C_VEL
LIN {X 0,Y 608.493,Z 324.086,A -85,B 0,C 180,E1 -461.186,E2 -461.186} C_VEL
LIN {X 0,Y 608.549,Z 311.281,A -85,B 0,C 180,E1 -461.554,E2 -461.554} C_VEL
LIN {X 0,Y 608.438,Z 300.493,A -85,B 0,C 180,E1 -461.767,E2 -461.767} C_VEL
LIN {X 0,Y 608.415,Z 291.936,A -85,B 0,C 180,E1 -464.38,E2 -464.38} C_VEL
LIN {X 0,Y 608.451,Z 284.145,A -85,B 0,C 180,E1 -466.784,E2 -466.784} C_VEL
LIN {X 0,Y 608.457,Z 275.241,A -85,B 0,C 180,E1 -469.57,E2 -469.57} C_VEL
LIN {X 0,Y 608.445,Z 266.13,A -85,B 0,C 180,E1 -472.472,E2 -472.472} C_VEL
LIN {X 0,Y 608.431,Z 258.545,A -85,B 0,C 180,E1 -474.936,E2 -474.936} C_VEL
LIN {X 0,Y 608.468,Z 250.754,A -85,B 0,C 180,E1 -477.516,E2 -477.516} C_VEL
LIN {X 0,Y 608.47,Z 243.471,A -85,B 0,C 180,E1 -479.971,E2 -479.971} C_VEL
LIN {X 0,Y 608.486,Z 236.091,A -85,B 0,C 180,E1 -482.525,E2 -482.525} C_VEL
LIN {X 0,Y 608.514,Z 227.958,A -85,B 0,C 180,E1 -485.475,E2 -485.475} C_VEL
LIN {X 0,Y 608.479,Z 227.693,A -85,B 0,C 180,E1 -485.681,E2 -485.681} C_VEL
LIN {X 0,Y 608.467,Z 227.696,A -85,B 0,C 180,E1 -488.24,E2 -488.24} C_VEL
LIN {X 0,Y 608.461,Z 227.697,A -85,B 0,C 180,E1 -491.342,E2 -491.342} C_VEL
LIN {X 0,Y 608.464,Z 227.694,A -85,B 0,C 180,E1 -493.869,E2 -493.869} C_VEL
LIN {X 0,Y 608.475,Z 227.694,A -85,B 0,C 180,E1 -496.689,E2 -496.689} C_VEL
LIN {X 0,Y 608.448,Z 227.698,A -85,B 0,C 180,E1 -499.67,E2 -499.67} C_VEL
LIN {X 0,Y 608.465,Z 227.694,A -85,B 0,C 180,E1 -502.253,E2 -502.253} C_VEL
LIN {X 0,Y 608.483,Z 227.692,A -85,B 0,C 180,E1 -505.088,E2 -505.088} C_VEL
LIN {X 0,Y 608.467,Z 227.695,A -85,B 0,C 180,E1 -507.905,E2 -507.905} C_VEL
LIN {X 0,Y 608.46,Z 227.695,A -85,B 0,C 180,E1 -510.219,E2 -510.219} C_VEL
LIN {X 0,Y 608.483,Z 227.694,A -85,B 0,C 180,E1 -512.79,E2 -512.79} C_VEL
LIN {X 0,Y 608.482,Z 227.694,A -85,B 0,C 180,E1 -515.844,E2 -515.844} C_VEL
LIN {X 0,Y 608.467,Z 227.694,A -85,B 0,C 180,E1 -518.308,E2 -518.308} C_VEL
LIN {X 0,Y 608.465,Z 227.695,A -85,B 0,C 180,E1 -521.282,E2 -521.282} C_VEL
LIN {X 0,Y 608.457,Z 227.695,A -85,B 0,C 180,E1 -523.905,E2 -523.905} C_VEL
LIN {X 0,Y 608.472,Z 227.693,A -85,B 0,C 180,E1 -526.643,E2 -526.643} C_VEL
LIN {X 0,Y 608.465,Z 227.697,A -85,B 0,C 180,E1 -529.349,E2 -529.349} C_VEL
LIN {X 0,Y 608.473,Z 227.693,A -85,B 0,C 180,E1 -532.032,E2 -532.032} C_VEL
LIN {X 0,Y 608.467,Z 227.694,A -85,B 0,C 180,E1 -534.697,E2 -534.697} C_VEL
LIN {X 0,Y 608.479,Z 227.693,A -85,B 0,C 180,E1 -537.351,E2 -537.351} C_VEL
LIN {X 0,Y 608.469,Z 227.693,A -85,B 0,C 180,E1 -539.999,E2 -539.999} C_VEL
LIN {X 0,Y 608.484,Z 227.695,A -85,B 0,C 180,E1 -542.647,E2 -542.647} C_VEL
LIN {X 0,Y 608.455,Z 227.695,A -85,B 0,C 180,E1 -545.301,E2 -545.301} C_VEL
LIN {X 0,Y 608.48,Z 227.693,A -85,B 0,C 180,E1 -547.966,E2 -547.966} C_VEL
LIN {X 0,Y 608.457,Z 227.694,A -85,B 0,C 180,E1 -549.475,E2 -549.475} C_VEL
LIN {X 0,Y 607.786,Z 227.899,A -85,B 0,C 180,E1 -550.027,E2 -550.027} C_VEL
LIN {X 0,Y 604.933,Z 228.923,A -85,B 0,C 180,E1 -550.918,E2 -550.918} C_VEL
LIN {X 0,Y 602.515,Z 230.123,A -85,B 0,C 180,E1 -551.633,E2 -551.633} C_VEL
LIN {X 0,Y 601.468,Z 231.111,A -85,B 0,C 180,E1 -552.182,E2 -552.182} C_VEL
LIN {X 0,Y 601.378,Z 231.439,A -85,B 0,C 180,E1 -552.369,E2 -552.369} C_VEL
LIN {X 0,Y 601.39,Z 235.852,A -85,B 0,C 180,E1 -554.897,E2 -554.897} C_VEL
LIN {X 0,Y 601.391,Z 240.817,A -85,B 0,C 180,E1 -557.687,E2 -557.687} C_VEL
LIN {X 0,Y 601.365,Z 245.923,A -85,B 0,C 180,E1 -560.523,E2 -560.523} C_VEL
LIN {X 0,Y 601.36,Z 251.369,A -85,B 0,C 180,E1 -563.412,E2 -563.412} C_VEL
LIN {X 0,Y 601.347,Z 257.057,A -85,B 0,C 180,E1 -566.365,E2 -566.365} C_VEL
LIN {X 0,Y 601.335,Z 263.004,A -85,B 0,C 180,E1 -569.396,E2 -569.396} C_VEL
LIN {X 0,Y 601.34,Z 269.231,A -85,B 0,C 180,E1 -572.52,E2 -572.52} C_VEL
LIN {X 0,Y 601.35,Z 272.576,A -85,B 0,C 180,E1 -574.173,E2 -574.173} C_VEL
LIN {X 0,Y 601.599,Z 283.057,A -85,B 0,C 180,E1 -574.397,E2 -574.397} C_VEL
LIN {X 0,Y 601.532,Z 295.262,A -85,B 0,C 180,E1 -574.77,E2 -574.77} C_VEL
LIN {X 0,Y 601.5,Z 307.948,A -85,B 0,C 180,E1 -575.308,E2 -575.308} C_VEL
LIN {X 0,Y 601.491,Z 319.195,A -85,B 0,C 180,E1 -575.928,E2 -575.928} C_VEL
LIN {X 0,Y 601.466,Z 330.058,A -85,B 0,C 180,E1 -576.681,E2 -576.681} C_VEL
LIN {X 0,Y 601.429,Z 339.829,A -85,B 0,C 180,E1 -577.524,E2 -577.524} C_VEL
LIN {X 0,Y 601.402,Z 348.772,A -85,B 0,C 180,E1 -578.469,E2 -578.469} C_VEL
LIN {X 0,Y 601.367,Z 356.795,A -85,B 0,C 180,E1 -579.529,E2 -579.529} C_VEL
LIN {X 0,Y 601.347,Z 363.07,A -85,B 0,C 180,E1 -580.567,E2 -580.567} C_VEL
LIN {X 0,Y 601.344,Z 368.718,A -85,B 0,C 180,E1 -581.77,E2 -581.77} C_VEL
LIN {X 0,Y 601.337,Z 371.894,A -85,B 0,C 180,E1 -582.675,E2 -582.675} C_VEL
LIN {X 0,Y 601.334,Z 374.311,A -85,B 0,C 180,E1 -583.593,E2 -583.593} C_VEL
LIN {X 0,Y 601.33,Z 376.515,A -85,B 0,C 180,E1 -584.997,E2 -584.997} C_VEL
LIN {X 0,Y 601.32,Z 376.852,A -85,B 0,C 180,E1 -585.473,E2 -585.473} C_VEL
LIN {X 0,Y 601.334,Z 376.916,A -85,B 0,C 180,E1 -586.435,E2 -586.435} C_VEL
LIN {X 0,Y 601.337,Z 376.148,A -85,B 0,C 180,E1 -587.415,E2 -587.415} C_VEL
LIN {X 0,Y 601.325,Z 374.484,A -85,B 0,C 180,E1 -588.416,E2 -588.416} C_VEL
LIN {X 0,Y 601.328,Z 371.832,A -85,B 0,C 180,E1 -589.435,E2 -589.435} C_VEL
LIN {X 0,Y 601.349,Z 368.07,A -85,B 0,C 180,E1 -590.473,E2 -590.473} C_VEL
LIN {X 0,Y 601.338,Z 362.987,A -85,B 0,C 180,E1 -591.538,E2 -591.538} C_VEL
LIN {X 0,Y 601.394,Z 356.395,A -85,B 0,C 180,E1 -592.621,E2 -592.621} C_VEL
LIN {X 0,Y 601.391,Z 348.926,A -85,B 0,C 180,E1 -593.604,E2 -593.604} C_VEL
LIN {X 0,Y 601.403,Z 339.548,A -85,B 0,C 180,E1 -594.594,E2 -594.594} C_VEL
LIN {X 0,Y 601.439,Z 329.175,A -85,B 0,C 180,E1 -595.478,E2 -595.478} C_VEL
LIN {X 0,Y 601.452,Z 318.418,A -85,B 0,C 180,E1 -596.21,E2 -596.21} C_VEL
LIN {X 0,Y 601.45,Z 306.532,A -85,B 0,C 180,E1 -596.852,E2 -596.852} C_VEL
LIN {X 0,Y 601.528,Z 294.645,A -85,B 0,C 180,E1 -597.343,E2 -597.343} C_VEL
LIN {X 0,Y 601.588,Z 281.485,A -85,B 0,C 180,E1 -597.73,E2 -597.73} C_VEL
LIN {X 0,Y 601.367,Z 273.389,A -85,B 0,C 180,E1 -597.902,E2 -597.902} C_VEL
LIN {X 0,Y 601.305,Z 272.55,A -85,B 0,C 180,E1 -597.923,E2 -597.923} C_VEL
LIN {X 0,Y 601.284,Z 267.17,A -85,B 0,C 180,E1 -600.6,E2 -600.6} C_VEL
LIN {X 0,Y 601.297,Z 262.634,A -85,B 0,C 180,E1 -602.882,E2 -602.882} C_VEL
LIN {X 0,Y 601.325,Z 257.052,A -85,B 0,C 180,E1 -605.728,E2 -605.728} C_VEL
LIN {X 0,Y 601.306,Z 252.597,A -85,B 0,C 180,E1 -608.037,E2 -608.037} C_VEL
LIN {X 0,Y 601.328,Z 248.509,A -85,B 0,C 180,E1 -610.188,E2 -610.188} C_VEL
LIN {X 0,Y 601.343,Z 244.543,A -85,B 0,C 180,E1 -612.31,E2 -612.31} C_VEL
LIN {X 0,Y 601.359,Z 239.508,A -85,B 0,C 180,E1 -615.102,E2 -615.102} C_VEL
LIN {X 0,Y 601.411,Z 234.63,A -85,B 0,C 180,E1 -617.858,E2 -617.858} C_VEL
LIN {X 0,Y 601.362,Z 229.898,A -85,B 0,C 180,E1 -620.583,E2 -620.583} C_VEL
LIN {X 0,Y 601.4,Z 228.737,A -85,B 0,C 180,E1 -621.262,E2 -621.262} C_VEL
LIN {X 0,Y 601.444,Z 228.568,A -85,B 0,C 180,E1 -623.324,E2 -623.324} C_VEL
LIN {X 0,Y 601.406,Z 228.576,A -85,B 0,C 180,E1 -625.98,E2 -625.98} C_VEL
LIN {X 0,Y 601.427,Z 228.571,A -85,B 0,C 180,E1 -628.661,E2 -628.661} C_VEL
LIN {X 0,Y 601.417,Z 228.571,A -85,B 0,C 180,E1 -631.339,E2 -631.339} C_VEL
LIN {X 0,Y 601.392,Z 228.574,A -85,B 0,C 180,E1 -634.021,E2 -634.021} C_VEL
LIN {X 0,Y 601.442,Z 228.57,A -85,B 0,C 180,E1 -636.71,E2 -636.71} C_VEL
LIN {X 0,Y 601.418,Z 228.572,A -85,B 0,C 180,E1 -639.416,E2 -639.416} C_VEL
LIN {X 0,Y 601.41,Z 228.572,A -85,B 0,C 180,E1 -642.142,E2 -642.142} C_VEL
LIN {X 0,Y 601.428,Z 228.57,A -85,B 0,C 180,E1 -644.897,E2 -644.897} C_VEL
LIN {X 0,Y 601.427,Z 228.569,A -85,B 0,C 180,E1 -646.986,E2 -646.986} C_VEL
LIN {X 0,Y 601.4,Z 228.575,A -85,B 0,C 180,E1 -649.809,E2 -649.809} C_VEL
LIN {X 0,Y 601.446,Z 228.568,A -85,B 0,C 180,E1 -652.681,E2 -652.681} C_VEL
LIN {X 0,Y 601.393,Z 228.577,A -85,B 0,C 180,E1 -654.879,E2 -654.879} C_VEL
LIN {X 0,Y 601.412,Z 228.574,A -85,B 0,C 180,E1 -657.365,E2 -657.365} C_VEL
LIN {X 0,Y 601.438,Z 228.568,A -85,B 0,C 180,E1 -660.163,E2 -660.163} C_VEL
LIN {X 0,Y 601.424,Z 228.57,A -85,B 0,C 180,E1 -662.718,E2 -662.718} C_VEL
LIN {X 0,Y 601.403,Z 228.572,A -85,B 0,C 180,E1 -665.115,E2 -665.115} C_VEL
LIN {X 0,Y 601.424,Z 228.57,A -85,B 0,C 180,E1 -667.419,E2 -667.419} C_VEL
LIN {X 0,Y 601.403,Z 228.573,A -85,B 0,C 180,E1 -669.995,E2 -669.995} C_VEL
LIN {X 0,Y 601.428,Z 228.571,A -85,B 0,C 180,E1 -672.668,E2 -672.668} C_VEL
LIN {X 0,Y 601.413,Z 228.572,A -85,B 0,C 180,E1 -675.482,E2 -675.482} C_VEL
LIN {X 0,Y 601.423,Z 228.57,A -85,B 0,C 180,E1 -678.406,E2 -678.406} C_VEL
LIN {X 0,Y 601.429,Z 228.57,A -85,B 0,C 180,E1 -680.876,E2 -680.876} C_VEL
LIN {X 0,Y 601.435,Z 228.571,A -85,B 0,C 180,E1 -683.734,E2 -683.734} C_VEL
LIN {X 0,Y 601.417,Z 228.571,A -85,B 0,C 180,E1 -686.687,E2 -686.687} C_VEL
LIN {X 0,Y 601.421,Z 228.57,A -85,B 0,C 180,E1 -689.059,E2 -689.059} C_VEL
LIN {X 0,Y 601.419,Z 228.571,A -85,B 0,C 180,E1 -691.374,E2 -691.374} C_VEL
LIN {X 0,Y 601.417,Z 228.572,A -85,B 0,C 180,E1 -694.13,E2 -694.13} C_VEL
LIN {X 0,Y 601.415,Z 228.572,A -85,B 0,C 180,E1 -696.591,E2 -696.591} C_VEL
LIN {X 0,Y 601.432,Z 228.57,A -85,B 0,C 180,E1 -699.479,E2 -699.479} C_VEL
LIN {X 0,Y 601.394,Z 228.574,A -85,B 0,C 180,E1 -702.313,E2 -702.313} C_VEL
LIN {X 0,Y 601.406,Z 228.573,A -85,B 0,C 180,E1 -704.41,E2 -704.41} C_VEL
LIN {X 0,Y 601.411,Z 228.572,A -85,B 0,C 180,E1 -707.173,E2 -707.173} C_VEL
LIN {X 0,Y 601.434,Z 228.571,A -85,B 0,C 180,E1 -709.906,E2 -709.906} C_VEL
LIN {X 0,Y 601.432,Z 228.571,A -85,B 0,C 180,E1 -712.616,E2 -712.616} C_VEL
LIN {X 0,Y 601.424,Z 228.57,A -85,B 0,C 180,E1 -715.309,E2 -715.309} C_VEL
LIN {X 0,Y 601.422,Z 228.57,A -85,B 0,C 180,E1 -717.992,E2 -717.992} C_VEL
LIN {X 0,Y 601.448,Z 228.569,A -85,B 0,C 180,E1 -720.67,E2 -720.67} C_VEL
LIN {X 0,Y 601.435,Z 228.571,A -85,B 0,C 180,E1 -723.35,E2 -723.35} C_VEL
LIN {X 0,Y 601.401,Z 228.573,A -85,B 0,C 180,E1 -726.038,E2 -726.038} C_VEL
LIN {X 0,Y 601.439,Z 228.572,A -85,B 0,C 180,E1 -728.062,E2 -728.062} C_VEL
LIN {X 0,Y 601.424,Z 228.57,A -85,B 0,C 180,E1 -731.017,E2 -731.017} C_VEL
LIN {X 0,Y 601.423,Z 228.57,A -85,B 0,C 180,E1 -733.516,E2 -733.516} C_VEL
LIN {X 0,Y 601.434,Z 228.571,A -85,B 0,C 180,E1 -736.288,E2 -736.288} C_VEL
LIN {X 0,Y 601.415,Z 228.572,A -85,B 0,C 180,E1 -739.1,E2 -739.1} C_VEL
LIN {X 0,Y 601.409,Z 228.572,A -85,B 0,C 180,E1 -741.96,E2 -741.96} C_VEL
LIN {X 0,Y 601.424,Z 228.57,A -85,B 0,C 180,E1 -744.292,E2 -744.292} C_VEL
LIN {X 0,Y 601.455,Z 228.568,A -85,B 0,C 180,E1 -747.112,E2 -747.112} C_VEL
LIN {X 0,Y 601.421,Z 228.572,A -85,B 0,C 180,E1 -749.394,E2 -749.394} C_VEL
LIN {X 0,Y 601.41,Z 228.573,A -85,B 0,C 180,E1 -751.727,E2 -751.727} C_VEL
LIN {X 0,Y 601.418,Z 228.572,A -85,B 0,C 180,E1 -754.12,E2 -754.12} C_VEL
LIN {X 0,Y 601.399,Z 228.574,A -85,B 0,C 180,E1 -756.584,E2 -756.584} C_VEL
LIN {X 0,Y 601.437,Z 228.571,A -85,B 0,C 180,E1 -759.125,E2 -759.125} C_VEL
LIN {X 0,Y 601.418,Z 228.573,A -85,B 0,C 180,E1 -761.766,E2 -761.766} C_VEL
LIN {X 0,Y 601.423,Z 228.57,A -85,B 0,C 180,E1 -764.536,E2 -764.536} C_VEL
LIN {X 0,Y 601.416,Z 228.572,A -85,B 0,C 180,E1 -767.409,E2 -767.409} C_VEL
LIN {X 0,Y 601.442,Z 228.568,A -85,B 0,C 180,E1 -770.465,E2 -770.465} C_VEL
LIN {X 0,Y 601.398,Z 228.575,A -85,B 0,C 180,E1 -773.417,E2 -773.417} C_VEL
LIN {X 0,Y 601.457,Z 228.732,A -85,B 0,C 180,E1 -774.337,E2 -774.337} C_VEL
LIN {X 0,Y 601.525,Z 235.119,A -85,B 0,C 180,E1 -776.693,E2 -776.693} C_VEL
LIN {X 0,Y 601.474,Z 242.898,A -85,B 0,C 180,E1 -779.451,E2 -779.451} C_VEL
LIN {X 0,Y 601.423,Z 250.752,A -85,B 0,C 180,E1 -782.133,E2 -782.133} C_VEL
LIN {X 0,Y 601.394,Z 258.545,A -85,B 0,C 180,E1 -784.752,E2 -784.752} C_VEL
LIN {X 0,Y 601.404,Z 266.584,A -85,B 0,C 180,E1 -787.398,E2 -787.398} C_VEL
LIN {X 0,Y 601.415,Z 275.24,A -85,B 0,C 180,E1 -790.191,E2 -790.191} C_VEL
LIN {X 0,Y 601.372,Z 284.144,A -85,B 0,C 180,E1 -793.013,E2 -793.013} C_VEL
LIN {X 0,Y 601.359,Z 293.049,A -85,B 0,C 180,E1 -795.793,E2 -795.793} C_VEL
LIN {X 0,Y 601.377,Z 300.492,A -85,B 0,C 180,E1 -798.092,E2 -798.092} C_VEL
LIN {X 0,Y 601.6,Z 313.937,A -85,B 0,C 180,E1 -798.374,E2 -798.374} C_VEL
LIN {X 0,Y 601.523,Z 326.342,A -85,B 0,C 180,E1 -798.766,E2 -798.766} C_VEL
LIN {X 0,Y 601.481,Z 338.926,A -85,B 0,C 180,E1 -799.31,E2 -799.31} C_VEL
LIN {X 0,Y 601.472,Z 349.582,A -85,B 0,C 180,E1 -799.906,E2 -799.906} C_VEL
LIN {X 0,Y 601.449,Z 360.477,A -85,B 0,C 180,E1 -800.669,E2 -800.669} C_VEL
LIN {X 0,Y 601.429,Z 371.113,A -85,B 0,C 180,E1 -801.601,E2 -801.601} C_VEL
LIN {X 0,Y 601.418,Z 378.961,A -85,B 0,C 180,E1 -802.446,E2 -802.446} C_VEL
LIN {X 0,Y 601.37,Z 386.226,A -85,B 0,C 180,E1 -803.398,E2 -803.398} C_VEL
LIN {X 0,Y 601.372,Z 391.866,A -85,B 0,C 180,E1 -804.299,E2 -804.299} C_VEL
LIN {X 0,Y 601.336,Z 396.95,A -85,B 0,C 180,E1 -805.307,E2 -805.307} C_VEL
LIN {X 0,Y 601.368,Z 400.896,A -85,B 0,C 180,E1 -806.315,E2 -806.315} C_VEL
LIN {X 0,Y 601.325,Z 403.809,A -85,B 0,C 180,E1 -807.32,E2 -807.32} C_VEL
LIN {X 0,Y 601.343,Z 405.202,A -85,B 0,C 180,E1 -807.991,E2 -807.991} C_VEL
LIN {X 0,Y 601.339,Z 406.784,A -85,B 0,C 180,E1 -809.33,E2 -809.33} C_VEL
LIN {X 0,Y 601.335,Z 407,A -85,B 0,C 180,E1 -810,E2 -810} C_VEL
LIN {X 0,Y 601.347,Z 406.184,A -85,B 0,C 180,E1 -811.339,E2 -811.339} C_VEL
LIN {X 0,Y 601.343,Z 405.202,A -85,B 0,C 180,E1 -812.009,E2 -812.009} C_VEL
LIN {X 0,Y 601.325,Z 403.81,A -85,B 0,C 180,E1 -812.679,E2 -812.679} C_VEL
LIN {X 0,Y 601.368,Z 400.897,A -85,B 0,C 180,E1 -813.685,E2 -813.685} C_VEL
LIN {X 0,Y 601.336,Z 396.951,A -85,B 0,C 180,E1 -814.692,E2 -814.692} C_VEL
LIN {X 0,Y 601.373,Z 390.878,A -85,B 0,C 180,E1 -815.869,E2 -815.869} C_VEL
LIN {X 0,Y 601.382,Z 384.237,A -85,B 0,C 180,E1 -816.88,E2 -816.88} C_VEL
LIN {X 0,Y 601.4,Z 375.992,A -85,B 0,C 180,E1 -817.892,E2 -817.892} C_VEL
LIN {X 0,Y 601.436,Z 367.54,A -85,B 0,C 180,E1 -818.737,E2 -818.737} C_VEL
LIN {X 0,Y 601.451,Z 357.096,A -85,B 0,C 180,E1 -819.585,E2 -819.585} C_VEL
LIN {X 0,Y 601.483,Z 346.762,A -85,B 0,C 180,E1 -820.264,E2 -820.264} C_VEL
LIN {X 0,Y 601.484,Z 335.223,A -85,B 0,C 180,E1 -820.869,E2 -820.869} C_VEL
LIN {X 0,Y 601.526,Z 322.343,A -85,B 0,C 180,E1 -821.375,E2 -821.375} C_VEL
LIN {X 0,Y 601.612,Z 309.452,A -85,B 0,C 180,E1 -821.732,E2 -821.732} C_VEL
LIN {X 0,Y 601.377,Z 300.493,A -85,B 0,C 180,E1 -821.908,E2 -821.908} C_VEL
LIN {X 0,Y 601.357,Z 291.936,A -85,B 0,C 180,E1 -824.552,E2 -824.552} C_VEL
LIN {X 0,Y 601.39,Z 283.032,A -85,B 0,C 180,E1 -827.337,E2 -827.337} C_VEL
LIN {X 0,Y 601.396,Z 274.128,A -85,B 0,C 180,E1 -830.165,E2 -830.165} C_VEL
LIN {X 0,Y 601.407,Z 265.223,A -85,B 0,C 180,E1 -833.046,E2 -833.046} C_VEL
LIN {X 0,Y 601.424,Z 256.679,A -85,B 0,C 180,E1 -835.869,E2 -835.869} C_VEL
LIN {X 0,Y 601.39,Z 248.441,A -85,B 0,C 180,E1 -838.628,E2 -838.628} C_VEL
LIN {X 0,Y 601.476,Z 241.742,A -85,B 0,C 180,E1 -840.938,E2 -840.938} C_VEL
LIN {X 0,Y 601.524,Z 235.083,A -85,B 0,C 180,E1 -843.307,E2 -843.307} C_VEL
LIN {X 0,Y 601.432,Z 228.572,A -85,B 0,C 180,E1 -845.751,E2 -845.751} C_VEL
LIN {X 0,Y 601.431,Z 228.571,A -85,B 0,C 180,E1 -848.47,E2 -848.47} C_VEL
LIN {X 0,Y 601.423,Z 228.572,A -85,B 0,C 180,E1 -851.592,E2 -851.592} C_VEL
LIN {X 0,Y 601.422,Z 228.573,A -85,B 0,C 180,E1 -854.534,E2 -854.534} C_VEL
LIN {X 0,Y 601.411,Z 228.575,A -85,B 0,C 180,E1 -857.408,E2 -857.408} C_VEL
LIN {X 0,Y 601.407,Z 228.573,A -85,B 0,C 180,E1 -860.004,E2 -860.004} C_VEL
LIN {X 0,Y 601.435,Z 228.573,A -85,B 0,C 180,E1 -862.616,E2 -862.616} C_VEL
LIN {X 0,Y 601.439,Z 228.569,A -85,B 0,C 180,E1 -865.069,E2 -865.069} C_VEL
LIN {X 0,Y 601.432,Z 228.571,A -85,B 0,C 180,E1 -867.484,E2 -867.484} C_VEL
LIN {X 0,Y 601.444,Z 228.571,A -85,B 0,C 180,E1 -869.847,E2 -869.847} C_VEL
LIN {X 0,Y 601.454,Z 228.57,A -85,B 0,C 180,E1 -872.888,E2 -872.888} C_VEL
LIN {X 0,Y 601.459,Z 228.568,A -85,B 0,C 180,E1 -875.859,E2 -875.859} C_VEL
LIN {X 0,Y 601.404,Z 228.574,A -85,B 0,C 180,E1 -878.76,E2 -878.76} C_VEL
LIN {X 0,Y 601.419,Z 228.571,A -85,B 0,C 180,E1 -881.608,E2 -881.608} C_VEL
LIN {X 0,Y 601.418,Z 228.573,A -85,B 0,C 180,E1 -884.408,E2 -884.408} C_VEL
LIN {X 0,Y 601.422,Z 228.573,A -85,B 0,C 180,E1 -887.171,E2 -887.171} C_VEL
LIN {X 0,Y 601.432,Z 228.57,A -85,B 0,C 180,E1 -889.904,E2 -889.904} C_VEL
LIN {X 0,Y 601.448,Z 228.569,A -85,B 0,C 180,E1 -892.614,E2 -892.614} C_VEL
LIN {X 0,Y 601.43,Z 228.571,A -85,B 0,C 180,E1 -895.307,E2 -895.307} C_VEL
LIN {X 0,Y 601.417,Z 228.572,A -85,B 0,C 180,E1 -897.99,E2 -897.99} C_VEL
LIN {X 0,Y 601.451,Z 228.57,A -85,B 0,C 180,E1 -900.669,E2 -900.669} C_VEL
LIN {X 0,Y 601.423,Z 228.572,A -85,B 0,C 180,E1 -903.349,E2 -903.349} C_VEL
LIN {X 0,Y 601.417,Z 228.572,A -85,B 0,C 180,E1 -906.036,E2 -906.036} C_VEL
LIN {X 0,Y 601.437,Z 228.572,A -85,B 0,C 180,E1 -908.737,E2 -908.737} C_VEL
LIN {X 0,Y 601.399,Z 228.69,A -85,B 0,C 180,E1 -910.776,E2 -910.776} C_VEL
LIN {X 0,Y 601.378,Z 231.439,A -85,B 0,C 180,E1 -912.369,E2 -912.369} C_VEL
LIN {X 0,Y 600.704,Z 232.476,A -85,B 0,C 180,E1 -912.919,E2 -912.919} C_VEL
LIN {X 0,Y 597.862,Z 234.354,A -85,B 0,C 180,E1 -913.81,E2 -913.81} C_VEL
LIN {X 0,Y 595.458,Z 235.863,A -85,B 0,C 180,E1 -914.526,E2 -914.526} C_VEL
LIN {X 0,Y 594.411,Z 236.93,A -85,B 0,C 180,E1 -915.08,E2 -915.08} C_VEL
LIN {X 0,Y 594.318,Z 237.265,A -85,B 0,C 180,E1 -915.268,E2 -915.268} C_VEL
LIN {X 0,Y 594.34,Z 241.94,A -85,B 0,C 180,E1 -917.904,E2 -917.904} C_VEL
LIN {X 0,Y 594.301,Z 247.216,A -85,B 0,C 180,E1 -920.9,E2 -920.9} C_VEL
LIN {X 0,Y 594.275,Z 252.463,A -85,B 0,C 180,E1 -923.708,E2 -923.708} C_VEL
LIN {X 0,Y 594.256,Z 258.18,A -85,B 0,C 180,E1 -926.705,E2 -926.705} C_VEL
LIN {X 0,Y 594.247,Z 262.638,A -85,B 0,C 180,E1 -929.004,E2 -929.004} C_VEL
LIN {X 0,Y 594.228,Z 267.779,A -85,B 0,C 180,E1 -931.621,E2 -931.621} C_VEL
LIN {X 0,Y 594.265,Z 272.529,A -85,B 0,C 180,E1 -934.014,E2 -934.014} C_VEL
LIN {X 0,Y 594.685,Z 278.17,A -85,B 0,C 180,E1 -934.144,E2 -934.144} C_VEL
LIN {X 0,Y 594.573,Z 291.328,A -85,B 0,C 180,E1 -934.501,E2 -934.501} C_VEL
LIN {X 0,Y 594.506,Z 303.777,A -85,B 0,C 180,E1 -934.983,E2 -934.983} C_VEL
LIN {X 0,Y 594.529,Z 315.831,A -85,B 0,C 180,E1 -935.603,E2 -935.603} C_VEL
LIN {X 0,Y 594.433,Z 325.625,A -85,B 0,C 180,E1 -936.237,E2 -936.237} C_VEL
LIN {X 0,Y 594.379,Z 336.215,A -85,B 0,C 180,E1 -937.086,E2 -937.086} C_VEL
LIN {X 0,Y 594.373,Z 344.912,A -85,B 0,C 180,E1 -937.94,E2 -937.94} C_VEL
LIN {X 0,Y 594.305,Z 352.231,A -85,B 0,C 180,E1 -938.81,E2 -938.81} C_VEL
LIN {X 0,Y 594.289,Z 359.836,A -85,B 0,C 180,E1 -939.93,E2 -939.93} C_VEL
LIN {X 0,Y 594.261,Z 366.125,A -85,B 0,C 180,E1 -941.116,E2 -941.116} C_VEL
LIN {X 0,Y 594.267,Z 369.171,A -85,B 0,C 180,E1 -941.837,E2 -941.837} C_VEL
LIN {X 0,Y 594.246,Z 372.523,A -85,B 0,C 180,E1 -942.841,E2 -942.841} C_VEL
LIN {X 0,Y 594.225,Z 374.865,A -85,B 0,C 180,E1 -943.826,E2 -943.826} C_VEL
LIN {X 0,Y 594.25,Z 376.67,A -85,B 0,C 180,E1 -945.201,E2 -945.201} C_VEL
LIN {X 0,Y 594.225,Z 376.977,A -85,B 0,C 180,E1 -946.173,E2 -946.173} C_VEL
LIN {X 0,Y 594.24,Z 376.462,A -85,B 0,C 180,E1 -947.159,E2 -947.159} C_VEL
LIN {X 0,Y 594.221,Z 374.316,A -85,B 0,C 180,E1 -948.524,E2 -948.524} C_VEL
LIN {X 0,Y 594.248,Z 371.99,A -85,B 0,C 180,E1 -949.424,E2 -949.424} C_VEL
LIN {X 0,Y 594.264,Z 368.953,A -85,B 0,C 180,E1 -950.312,E2 -950.312} C_VEL
LIN {X 0,Y 594.286,Z 364.549,A -85,B 0,C 180,E1 -951.306,E2 -951.306} C_VEL
LIN {X 0,Y 594.268,Z 358.336,A -85,B 0,C 180,E1 -952.405,E2 -952.405} C_VEL
LIN {X 0,Y 594.33,Z 350.309,A -85,B 0,C 180,E1 -953.522,E2 -953.522} C_VEL
LIN {X 0,Y 594.386,Z 341.665,A -85,B 0,C 180,E1 -954.49,E2 -954.49} C_VEL
LIN {X 0,Y 594.417,Z 331.262,A -85,B 0,C 180,E1 -955.423,E2 -955.423} C_VEL
LIN {X 0,Y 594.435,Z 320.946,A -85,B 0,C 180,E1 -956.172,E2 -956.172} C_VEL
LIN {X 0,Y 594.453,Z 311.078,A -85,B 0,C 180,E1 -956.752,E2 -956.752} C_VEL
LIN {X 0,Y 594.517,Z 299.005,A -85,B 0,C 180,E1 -957.311,E2 -957.311} C_VEL
LIN {X 0,Y 594.602,Z 285.84,A -85,B 0,C 180,E1 -957.755,E2 -957.755} C_VEL
LIN {X 0,Y 594.46,Z 274.242,A -85,B 0,C 180,E1 -958.026,E2 -958.026} C_VEL
LIN {X 0,Y 594.195,Z 272.554,A -85,B 0,C 180,E1 -958.065,E2 -958.065} C_VEL
LIN {X 0,Y 594.232,Z 266.6,A -85,B 0,C 180,E1 -961.066,E2 -961.066} C_VEL
LIN {X 0,Y 594.221,Z 260.765,A -85,B 0,C 180,E1 -964.049,E2 -964.049} C_VEL
LIN {X 0,Y 594.217,Z 256.447,A -85,B 0,C 180,E1 -966.289,E2 -966.289} C_VEL
LIN {X 0,Y 594.248,Z 252.257,A -85,B 0,C 180,E1 -968.493,E2 -968.493} C_VEL
LIN {X 0,Y 594.28,Z 246.869,A -85,B 0,C 180,E1 -971.38,E2 -971.38} C_VEL
LIN {X 0,Y 594.297,Z 243.072,A -85,B 0,C 180,E1 -973.512,E2 -973.512} C_VEL
LIN {X 0,Y 594.335,Z 238.069,A -85,B 0,C 180,E1 -976.32,E2 -976.32} C_VEL
LIN {X 0,Y 594.372,Z 233.244,A -85,B 0,C 180,E1 -979.095,E2 -979.095} C_VEL
LIN {X 0,Y 594.335,Z 229.742,A -85,B 0,C 180,E1 -981.157,E2 -981.157} C_VEL
LIN {X 0,Y 594.394,Z 229.448,A -85,B 0,C 180,E1 -982.527,E2 -982.527} C_VEL
LIN {X 0,Y 594.386,Z 229.447,A -85,B 0,C 180,E1 -985.253,E2 -985.253} C_VEL
LIN {X 0,Y 594.382,Z 229.447,A -85,B 0,C 180,E1 -987.967,E2 -987.967} C_VEL
LIN {X 0,Y 594.418,Z 229.445,A -85,B 0,C 180,E1 -990.678,E2 -990.678} C_VEL
LIN {X 0,Y 594.381,Z 229.449,A -85,B 0,C 180,E1 -993.389,E2 -993.389} C_VEL
LIN {X 0,Y 594.356,Z 229.45,A -85,B 0,C 180,E1 -996.109,E2 -996.109} C_VEL
LIN {X 0,Y 594.395,Z 229.446,A -85,B 0,C 180,E1 -998.842,E2 -998.842} C_VEL
LIN {X 0,Y 594.386,Z 229.45,A -85,B 0,C 180,E1 -1001.596,E2 -1001.596} C_VEL
LIN {X 0,Y 594.381,Z 229.448,A -85,B 0,C 180,E1 -1004.377,E2 -1004.377} C_VEL
LIN {X 0,Y 594.383,Z 229.447,A -85,B 0,C 180,E1 -1007.193,E2 -1007.193} C_VEL
LIN {X 0,Y 594.371,Z 229.452,A -85,B 0,C 180,E1 -1010.054,E2 -1010.054} C_VEL
LIN {X 0,Y 594.389,Z 229.446,A -85,B 0,C 180,E1 -1012.966,E2 -1012.966} C_VEL
LIN {X 0,Y 594.364,Z 229.45,A -85,B 0,C 180,E1 -1015.193,E2 -1015.193} C_VEL
LIN {X 0,Y 594.373,Z 229.449,A -85,B 0,C 180,E1 -1017.527,E2 -1017.527} C_VEL
LIN {X 0,Y 594.39,Z 229.446,A -85,B 0,C 180,E1 -1020.331,E2 -1020.331} C_VEL
LIN {X 0,Y 594.37,Z 229.449,A -85,B 0,C 180,E1 -1022.95,E2 -1022.95} C_VEL
LIN {X 0,Y 594.373,Z 229.45,A -85,B 0,C 180,E1 -1025.407,E2 -1025.407} C_VEL
LIN {X 0,Y 594.382,Z 229.45,A -85,B 0,C 180,E1 -1027.94,E2 -1027.94} C_VEL
LIN {X 0,Y 594.376,Z 229.448,A -85,B 0,C 180,E1 -1030.824,E2 -1030.824} C_VEL
LIN {X 0,Y 594.374,Z 229.448,A -85,B 0,C 180,E1 -1033.298,E2 -1033.298} C_VEL
LIN {X 0,Y 594.37,Z 229.45,A -85,B 0,C 180,E1 -1036.159,E2 -1036.159} C_VEL
LIN {X 0,Y 594.379,Z 229.448,A -85,B 0,C 180,E1 -1038.538,E2 -1038.538} C_VEL
LIN {X 0,Y 594.38,Z 229.45,A -85,B 0,C 180,E1 -1041.295,E2 -1041.295} C_VEL
LIN {X 0,Y 594.387,Z 229.449,A -85,B 0,C 180,E1 -1043.759,E2 -1043.759} C_VEL
LIN {X 0,Y 594.369,Z 229.45,A -85,B 0,C 180,E1 -1046.239,E2 -1046.239} C_VEL
LIN {X 0,Y 594.381,Z 229.449,A -85,B 0,C 180,E1 -1048.652,E2 -1048.652} C_VEL
LIN {X 0,Y 594.372,Z 229.45,A -85,B 0,C 180,E1 -1051.042,E2 -1051.042} C_VEL
LIN {X 0,Y 594.389,Z 229.446,A -85,B 0,C 180,E1 -1053.975,E2 -1053.975} C_VEL
LIN {X 0,Y 594.388,Z 229.446,A -85,B 0,C 180,E1 -1056.297,E2 -1056.297} C_VEL
LIN {X 0,Y 594.402,Z 229.448,A -85,B 0,C 180,E1 -1059.225,E2 -1059.225} C_VEL
LIN {X 0,Y 594.373,Z 229.448,A -85,B 0,C 180,E1 -1062.097,E2 -1062.097} C_VEL
LIN {X 0,Y 594.362,Z 229.451,A -85,B 0,C 180,E1 -1064.22,E2 -1064.22} C_VEL
LIN {X 0,Y 594.358,Z 229.45,A -85,B 0,C 180,E1 -1067.018,E2 -1067.018} C_VEL
LIN {X 0,Y 594.393,Z 229.447,A -85,B 0,C 180,E1 -1069.785,E2 -1069.785} C_VEL
LIN {X 0,Y 594.386,Z 229.449,A -85,B 0,C 180,E1 -1072.528,E2 -1072.528} C_VEL
LIN {X 0,Y 594.392,Z 229.446,A -85,B 0,C 180,E1 -1075.253,E2 -1075.253} C_VEL
LIN {X 0,Y 594.392,Z 229.446,A -85,B 0,C 180,E1 -1077.968,E2 -1077.968} C_VEL
LIN {X 0,Y 594.419,Z 229.445,A -85,B 0,C 180,E1 -1080.678,E2 -1080.678} C_VEL
LIN {X 0,Y 594.385,Z 229.449,A -85,B 0,C 180,E1 -1083.39,E2 -1083.39} C_VEL
LIN {X 0,Y 594.358,Z 229.45,A -85,B 0,C 180,E1 -1086.11,E2 -1086.11} C_VEL
LIN {X 0,Y 594.41,Z 229.446,A -85,B 0,C 180,E1 -1088.157,E2 -1088.157} C_VEL
LIN {X 0,Y 594.388,Z 229.446,A -85,B 0,C 180,E1 -1091.078,E2 -1091.078} C_VEL
LIN {X 0,Y 594.384,Z 229.447,A -85,B 0,C 180,E1 -1093.68,E2 -1093.68} C_VEL
LIN {X 0,Y 594.394,Z 229.446,A -85,B 0,C 180,E1 -1096.722,E2 -1096.722} C_VEL
LIN {X 0,Y 594.366,Z 229.449,A -85,B 0,C 180,E1 -1099.335,E2 -1099.335} C_VEL
LIN {X 0,Y 594.36,Z 229.451,A -85,B 0,C 180,E1 -1101.504,E2 -1101.504} C_VEL
LIN {X 0,Y 594.384,Z 229.447,A -85,B 0,C 180,E1 -1104.447,E2 -1104.447} C_VEL
LIN {X 0,Y 594.384,Z 229.447,A -85,B 0,C 180,E1 -1106.7,E2 -1106.7} C_VEL
LIN {X 0,Y 594.384,Z 229.447,A -85,B 0,C 180,E1 -1108.999,E2 -1108.999} C_VEL
LIN {X 0,Y 594.388,Z 229.447,A -85,B 0,C 180,E1 -1111.646,E2 -1111.646} C_VEL
LIN {X 0,Y 594.393,Z 229.448,A -85,B 0,C 180,E1 -1114.58,E2 -1114.58} C_VEL
LIN {X 0,Y 594.388,Z 229.447,A -85,B 0,C 180,E1 -1117.609,E2 -1117.609} C_VEL
LIN {X 0,Y 594.369,Z 229.451,A -85,B 0,C 180,E1 -1120.568,E2 -1120.568} C_VEL
LIN {X 0,Y 594.363,Z 229.45,A -85,B 0,C 180,E1 -1123.3,E2 -1123.3} C_VEL
LIN {X 0,Y 594.359,Z 229.451,A -85,B 0,C 180,E1 -1126.162,E2 -1126.162} C_VEL
LIN {X 0,Y 594.381,Z 229.448,A -85,B 0,C 180,E1 -1128.537,E2 -1128.537} C_VEL
LIN {X 0,Y 594.378,Z 229.451,A -85,B 0,C 180,E1 -1131.297,E2 -1131.297} C_VEL
LIN {X 0,Y 594.407,Z 229.594,A -85,B 0,C 180,E1 -1134.179,E2 -1134.179} C_VEL
LIN {X 0,Y 594.51,Z 235.103,A -85,B 0,C 180,E1 -1136.248,E2 -1136.248} C_VEL
LIN {X 0,Y 594.467,Z 242.86,A -85,B 0,C 180,E1 -1139.052,E2 -1139.052} C_VEL
LIN {X 0,Y 594.379,Z 250.637,A -85,B 0,C 180,E1 -1141.774,E2 -1141.774} C_VEL
LIN {X 0,Y 594.403,Z 258.545,A -85,B 0,C 180,E1 -1144.434,E2 -1144.434} C_VEL
LIN {X 0,Y 594.353,Z 267.05,A -85,B 0,C 180,E1 -1147.268,E2 -1147.268} C_VEL
LIN {X 0,Y 594.339,Z 275.24,A -85,B 0,C 180,E1 -1149.945,E2 -1149.945} C_VEL
LIN {X 0,Y 594.317,Z 284.144,A -85,B 0,C 180,E1 -1152.805,E2 -1152.805} C_VEL
LIN {X 0,Y 594.295,Z 293.049,A -85,B 0,C 180,E1 -1155.621,E2 -1155.621} C_VEL
LIN {X 0,Y 594.286,Z 300.492,A -85,B 0,C 180,E1 -1157.948,E2 -1157.948} C_VEL
LIN {X 0,Y 594.673,Z 305.237,A -85,B 0,C 180,E1 -1158.042,E2 -1158.042} C_VEL
LIN {X 0,Y 594.613,Z 318.501,A -85,B 0,C 180,E1 -1158.366,E2 -1158.366} C_VEL
LIN {X 0,Y 594.532,Z 330.65,A -85,B 0,C 180,E1 -1158.801,E2 -1158.801} C_VEL
LIN {X 0,Y 594.478,Z 342.212,A -85,B 0,C 180,E1 -1159.355,E2 -1159.355} C_VEL
LIN {X 0,Y 594.471,Z 353.479,A -85,B 0,C 180,E1 -1160.044,E2 -1160.044} C_VEL
LIN {X 0,Y 594.406,Z 363.648,A -85,B 0,C 180,E1 -1160.815,E2 -1160.815} C_VEL
LIN {X 0,Y 594.372,Z 372.788,A -85,B 0,C 180,E1 -1161.672,E2 -1161.672} C_VEL
LIN {X 0,Y 594.317,Z 381.691,A -85,B 0,C 180,E1 -1162.697,E2 -1162.697} C_VEL
LIN {X 0,Y 594.281,Z 388.171,A -85,B 0,C 180,E1 -1163.615,E2 -1163.615} C_VEL
LIN {X 0,Y 594.289,Z 393.68,A -85,B 0,C 180,E1 -1164.571,E2 -1164.571} C_VEL
LIN {X 0,Y 594.27,Z 398.371,A -85,B 0,C 180,E1 -1165.591,E2 -1165.591} C_VEL
LIN {X 0,Y 594.267,Z 401.956,A -85,B 0,C 180,E1 -1166.61,E2 -1166.61} C_VEL
LIN {X 0,Y 594.226,Z 403.809,A -85,B 0,C 180,E1 -1167.288,E2 -1167.288} C_VEL
LIN {X 0,Y 594.242,Z 405.201,A -85,B 0,C 180,E1 -1167.967,E2 -1167.967} C_VEL
LIN {X 0,Y 594.239,Z 406.784,A -85,B 0,C 180,E1 -1169.322,E2 -1169.322} C_VEL
LIN {X 0,Y 594.236,Z 407,A -85,B 0,C 180,E1 -1170,E2 -1170} C_VEL
LIN {X 0,Y 594.247,Z 406.185,A -85,B 0,C 180,E1 -1171.355,E2 -1171.355} C_VEL
LIN {X 0,Y 594.242,Z 405.202,A -85,B 0,C 180,E1 -1172.033,E2 -1172.033} C_VEL
LIN {X 0,Y 594.226,Z 403.81,A -85,B 0,C 180,E1 -1172.711,E2 -1172.711} C_VEL
LIN {X 0,Y 594.289,Z 400.897,A -85,B 0,C 180,E1 -1173.729,E2 -1173.729} C_VEL
LIN {X 0,Y 594.241,Z 396.95,A -85,B 0,C 180,E1 -1174.749,E2 -1174.749} C_VEL
LIN {X 0,Y 594.305,Z 390.879,A -85,B 0,C 180,E1 -1175.939,E2 -1175.939} C_VEL
LIN {X 0,Y 594.308,Z 384.238,A -85,B 0,C 180,E1 -1176.962,E2 -1176.962} C_VEL
LIN {X 0,Y 594.359,Z 375.992,A -85,B 0,C 180,E1 -1177.986,E2 -1177.986} C_VEL
LIN {X 0,Y 594.382,Z 367.54,A -85,B 0,C 180,E1 -1178.842,E2 -1178.842} C_VEL
LIN {X 0,Y 594.435,Z 357.098,A -85,B 0,C 180,E1 -1179.699,E2 -1179.699} C_VEL
LIN {X 0,Y 594.458,Z 346.764,A -85,B 0,C 180,E1 -1180.387,E2 -1180.387} C_VEL
LIN {X 0,Y 594.502,Z 334.776,A -85,B 0,C 180,E1 -1181.019,E2 -1181.019} C_VEL
LIN {X 0,Y 594.564,Z 322.499,A -85,B 0,C 180,E1 -1181.505,E2 -1181.505} C_VEL
LIN {X 0,Y 594.684,Z 309.451,A -85,B 0,C 180,E1 -1181.871,E2 -1181.871} C_VEL
LIN {X 0,Y 594.425,Z 301.636,A -85,B 0,C 180,E1 -1182.027,E2 -1182.027} C_VEL
LIN {X 0,Y 594.291,Z 300.423,A -85,B 0,C 180,E1 -1182.073,E2 -1182.073} C_VEL
LIN {X 0,Y 594.3,Z 291.936,A -85,B 0,C 180,E1 -1184.729,E2 -1184.729} C_VEL
LIN {X 0,Y 594.325,Z 283.032,A -85,B 0,C 180,E1 -1187.55,E2 -1187.55} C_VEL
LIN {X 0,Y 594.357,Z 274.128,A -85,B 0,C 180,E1 -1190.415,E2 -1190.415} C_VEL
LIN {X 0,Y 594.36,Z 265.223,A -85,B 0,C 180,E1 -1193.335,E2 -1193.335} C_VEL
LIN {X 0,Y 594.392,Z 257.195,A -85,B 0,C 180,E1 -1196.023,E2 -1196.023} C_VEL
LIN {X 0,Y 594.369,Z 249.513,A -85,B 0,C 180,E1 -1198.591,E2 -1198.591} C_VEL
LIN {X 0,Y 594.466,Z 242.808,A -85,B 0,C 180,E1 -1200.948,E2 -1200.948} C_VEL
LIN {X 0,Y 594.5,Z 235.062,A -85,B 0,C 180,E1 -1203.753,E2 -1203.753} C_VEL
LIN {X 0,Y 594.421,Z 229.6,A -85,B 0,C 180,E1 -1205.82,E2 -1205.82} C_VEL
LIN {X 0,Y 594.377,Z 229.449,A -85,B 0,C 180,E1 -1208.805,E2 -1208.805} C_VEL
LIN {X 0,Y 594.381,Z 229.448,A -85,B 0,C 180,E1 -1211.848,E2 -1211.848} C_VEL
LIN {X 0,Y 594.38,Z 229.45,A -85,B 0,C 180,E1 -1214.235,E2 -1214.235} C_VEL
LIN {X 0,Y 594.36,Z 229.451,A -85,B 0,C 180,E1 -1217.147,E2 -1217.147} C_VEL
LIN {X 0,Y 594.37,Z 229.452,A -85,B 0,C 180,E1 -1219.432,E2 -1219.432} C_VEL
LIN {X 0,Y 594.388,Z 229.448,A -85,B 0,C 180,E1 -1222.39,E2 -1222.39} C_VEL
LIN {X 0,Y 594.382,Z 229.451,A -85,B 0,C 180,E1 -1224.671,E2 -1224.671} C_VEL
LIN {X 0,Y 594.377,Z 229.449,A -85,B 0,C 180,E1 -1227.087,E2 -1227.087} C_VEL
LIN {X 0,Y 594.397,Z 229.448,A -85,B 0,C 180,E1 -1229.668,E2 -1229.668} C_VEL
LIN {X 0,Y 594.386,Z 229.448,A -85,B 0,C 180,E1 -1232.539,E2 -1232.539} C_VEL
LIN {X 0,Y 594.392,Z 229.447,A -85,B 0,C 180,E1 -1235.563,E2 -1235.563} C_VEL
LIN {X 0,Y 594.363,Z 229.45,A -85,B 0,C 180,E1 -1238.496,E2 -1238.496} C_VEL
LIN {X 0,Y 594.382,Z 229.449,A -85,B 0,C 180,E1 -1241.382,E2 -1241.382} C_VEL
LIN {X 0,Y 594.369,Z 229.452,A -85,B 0,C 180,E1 -1244.218,E2 -1244.218} C_VEL
LIN {X 0,Y 594.37,Z 229.45,A -85,B 0,C 180,E1 -1247.016,E2 -1247.016} C_VEL
LIN {X 0,Y 594.392,Z 229.447,A -85,B 0,C 180,E1 -1249.783,E2 -1249.783} C_VEL
LIN {X 0,Y 594.396,Z 229.448,A -85,B 0,C 180,E1 -1252.526,E2 -1252.526} C_VEL
LIN {X 0,Y 594.398,Z 229.447,A -85,B 0,C 180,E1 -1255.252,E2 -1255.252} C_VEL
LIN {X 0,Y 594.387,Z 229.447,A -85,B 0,C 180,E1 -1257.966,E2 -1257.966} C_VEL
LIN {X 0,Y 594.421,Z 229.445,A -85,B 0,C 180,E1 -1260.677,E2 -1260.677} C_VEL
LIN {X 0,Y 594.375,Z 229.45,A -85,B 0,C 180,E1 -1263.389,E2 -1263.389} C_VEL
LIN {X 0,Y 594.372,Z 229.45,A -85,B 0,C 180,E1 -1266.108,E2 -1266.108} C_VEL
LIN {X 0,Y 594.397,Z 229.449,A -85,B 0,C 180,E1 -1268.841,E2 -1268.841} C_VEL
LIN {X 0,Y 594.376,Z 229.45,A -85,B 0,C 180,E1 -1270.215,E2 -1270.215} C_VEL
LIN {X 0,Y 594.378,Z 230.035,A -85,B 0,C 180,E1 -1271.074,E2 -1271.074} C_VEL
LIN {X 0,Y 594.348,Z 235.729,A -85,B 0,C 180,E1 -1274.377,E2 -1274.377} C_VEL
LIN {X 0,Y 594.318,Z 237.265,A -85,B 0,C 180,E1 -1275.268,E2 -1275.268} C_VEL
LIN {X 0,Y 593.634,Z 238.311,A -85,B 0,C 180,E1 -1275.824,E2 -1275.824} C_VEL
LIN {X 0,Y 590.789,Z 240.205,A -85,B 0,C 180,E1 -1276.725,E2 -1276.725} C_VEL
LIN {X 0,Y 588.39,Z 241.741,A -85,B 0,C 180,E1 -1277.448,E2 -1277.448} C_VEL
LIN {X 0,Y 587.351,Z 242.845,A -85,B 0,C 180,E1 -1278.008,E2 -1278.008} C_VEL
LIN {X 0,Y 587.261,Z 243.193,A -85,B 0,C 180,E1 -1278.198,E2 -1278.198} C_VEL
LIN {X 0,Y 587.229,Z 248.115,A -85,B 0,C 180,E1 -1281.04,E2 -1281.04} C_VEL
LIN {X 0,Y 587.193,Z 252.165,A -85,B 0,C 180,E1 -1283.263,E2 -1283.263} C_VEL
LIN {X 0,Y 587.199,Z 257.589,A -85,B 0,C 180,E1 -1286.152,E2 -1286.152} C_VEL
LIN {X 0,Y 587.159,Z 263.235,A -85,B 0,C 180,E1 -1289.102,E2 -1289.102} C_VEL
LIN {X 0,Y 587.133,Z 268.484,A -85,B 0,C 180,E1 -1291.804,E2 -1291.804} C_VEL
LIN {X 0,Y 587.178,Z 272.534,A -85,B 0,C 180,E1 -1293.869,E2 -1293.869} C_VEL
LIN {X 0,Y 587.706,Z 277.596,A -85,B 0,C 180,E1 -1293.989,E2 -1293.989} C_VEL
LIN {X 0,Y 587.636,Z 289.9,A -85,B 0,C 180,E1 -1294.315,E2 -1294.315} C_VEL
LIN {X 0,Y 587.569,Z 302.422,A -85,B 0,C 180,E1 -1294.79,E2 -1294.79} C_VEL
LIN {X 0,Y 587.503,Z 314.541,A -85,B 0,C 180,E1 -1295.402,E2 -1295.402} C_VEL
LIN {X 0,Y 587.422,Z 325.381,A -85,B 0,C 180,E1 -1296.101,E2 -1296.101} C_VEL
LIN {X 0,Y 587.364,Z 336.001,A -85,B 0,C 180,E1 -1296.959,E2 -1296.959} C_VEL
LIN {X 0,Y 587.326,Z 344.875,A -85,B 0,C 180,E1 -1297.838,E2 -1297.838} C_VEL
LIN {X 0,Y 587.232,Z 352.141,A -85,B 0,C 180,E1 -1298.711,E2 -1298.711} C_VEL
LIN {X 0,Y 587.224,Z 358.831,A -85,B 0,C 180,E1 -1299.686,E2 -1299.686} C_VEL
LIN {X 0,Y 587.175,Z 364.255,A -85,B 0,C 180,E1 -1300.66,E2 -1300.66} C_VEL
LIN {X 0,Y 587.17,Z 368.552,A -85,B 0,C 180,E1 -1301.627,E2 -1301.627} C_VEL
LIN {X 0,Y 587.162,Z 373.086,A -85,B 0,C 180,E1 -1303.019,E2 -1303.019} C_VEL
LIN {X 0,Y 587.142,Z 375.378,A -85,B 0,C 180,E1 -1304.096,E2 -1304.096} C_VEL
LIN {X 0,Y 587.171,Z 376.591,A -85,B 0,C 180,E1 -1305.076,E2 -1305.076} C_VEL
LIN {X 0,Y 587.124,Z 377,A -85,B 0,C 180,E1 -1306.032,E2 -1306.032} C_VEL
LIN {X 0,Y 587.155,Z 376.614,A -85,B 0,C 180,E1 -1306.98,E2 -1306.98} C_VEL
LIN {X 0,Y 587.149,Z 375.51,A -85,B 0,C 180,E1 -1307.911,E2 -1307.911} C_VEL
LIN {X 0,Y 587.125,Z 373.406,A -85,B 0,C 180,E1 -1308.947,E2 -1308.947} C_VEL
LIN {X 0,Y 587.183,Z 370.28,A -85,B 0,C 180,E1 -1309.996,E2 -1309.996} C_VEL
LIN {X 0,Y 587.205,Z 364.9,A -85,B 0,C 180,E1 -1311.294,E2 -1311.294} C_VEL
LIN {X 0,Y 587.184,Z 358.972,A -85,B 0,C 180,E1 -1312.381,E2 -1312.381} C_VEL
LIN {X 0,Y 587.269,Z 351.275,A -85,B 0,C 180,E1 -1313.489,E2 -1313.489} C_VEL
LIN {X 0,Y 587.297,Z 342.921,A -85,B 0,C 180,E1 -1314.46,E2 -1314.46} C_VEL
LIN {X 0,Y 587.386,Z 333.787,A -85,B 0,C 180,E1 -1315.328,E2 -1315.328} C_VEL
LIN {X 0,Y 587.436,Z 323.859,A -85,B 0,C 180,E1 -1316.096,E2 -1316.096} C_VEL
LIN {X 0,Y 587.464,Z 312.992,A -85,B 0,C 180,E1 -1316.775,E2 -1316.775} C_VEL
LIN {X 0,Y 587.513,Z 301.501,A -85,B 0,C 180,E1 -1317.342,E2 -1317.342} C_VEL
LIN {X 0,Y 587.637,Z 289.283,A -85,B 0,C 180,E1 -1317.796,E2 -1317.796} C_VEL
LIN {X 0,Y 587.729,Z 276.595,A -85,B 0,C 180,E1 -1318.12,E2 -1318.12} C_VEL
LIN {X 0,Y 587.132,Z 272.54,A -85,B 0,C 180,E1 -1318.219,E2 -1318.219} C_VEL
LIN {X 0,Y 587.14,Z 267.283,A -85,B 0,C 180,E1 -1320.901,E2 -1320.901} C_VEL
LIN {X 0,Y 587.144,Z 261.56,A -85,B 0,C 180,E1 -1323.859,E2 -1323.859} C_VEL
LIN {X 0,Y 587.16,Z 257.501,A -85,B 0,C 180,E1 -1325.986,E2 -1325.986} C_VEL
LIN {X 0,Y 587.154,Z 253.299,A -85,B 0,C 180,E1 -1328.22,E2 -1328.22} C_VEL
LIN {X 0,Y 587.226,Z 248.201,A -85,B 0,C 180,E1 -1330.99,E2 -1330.99} C_VEL
LIN {X 0,Y 587.216,Z 242.86,A -85,B 0,C 180,E1 -1334.022,E2 -1334.022} C_VEL
LIN {X 0,Y 587.255,Z 237.888,A -85,B 0,C 180,E1 -1336.857,E2 -1336.857} C_VEL
LIN {X 0,Y 587.297,Z 233.072,A -85,B 0,C 180,E1 -1339.66,E2 -1339.66} C_VEL
LIN {X 0,Y 587.276,Z 230.745,A -85,B 0,C 180,E1 -1341.05,E2 -1341.05} C_VEL
LIN {X 0,Y 587.328,Z 230.324,A -85,B 0,C 180,E1 -1341.744,E2 -1341.744} C_VEL
LIN {X 0,Y 587.353,Z 230.324,A -85,B 0,C 180,E1 -1344.507,E2 -1344.507} C_VEL
LIN {X 0,Y 587.368,Z 230.324,A -85,B 0,C 180,E1 -1347.257,E2 -1347.257} C_VEL
LIN {X 0,Y 587.369,Z 230.321,A -85,B 0,C 180,E1 -1350,E2 -1350} C_VEL
LIN {X 0,Y 587.369,Z 230.321,A -85,B 0,C 180,E1 -1352.743,E2 -1352.743} C_VEL
LIN {X 0,Y 587.353,Z 230.325,A -85,B 0,C 180,E1 -1355.493,E2 -1355.493} C_VEL
LIN {X 0,Y 587.365,Z 230.323,A -85,B 0,C 180,E1 -1358.255,E2 -1358.255} C_VEL
LIN {X 0,Y 587.352,Z 230.323,A -85,B 0,C 180,E1 -1361.141,E2 -1361.141} C_VEL
LIN {X 0,Y 587.354,Z 230.324,A -85,B 0,C 180,E1 -1364.261,E2 -1364.261} C_VEL
LIN {X 0,Y 587.349,Z 230.324,A -85,B 0,C 180,E1 -1367.406,E2 -1367.406} C_VEL
LIN {X 0,Y 587.327,Z 230.327,A -85,B 0,C 180,E1 -1370.305,E2 -1370.305} C_VEL
LIN {X 0,Y 587.357,Z 230.322,A -85,B 0,C 180,E1 -1373.257,E2 -1373.257} C_VEL
LIN {X 0,Y 587.352,Z 230.324,A -85,B 0,C 180,E1 -1376.277,E2 -1376.277} C_VEL
LIN {X 0,Y 587.345,Z 230.324,A -85,B 0,C 180,E1 -1379.135,E2 -1379.135} C_VEL
LIN {X 0,Y 587.348,Z 230.325,A -85,B 0,C 180,E1 -1381.838,E2 -1381.838} C_VEL
LIN {X 0,Y 587.341,Z 230.327,A -85,B 0,C 180,E1 -1384.349,E2 -1384.349} C_VEL
LIN {X 0,Y 587.343,Z 230.327,A -85,B 0,C 180,E1 -1386.747,E2 -1386.747} C_VEL
LIN {X 0,Y 587.337,Z 230.327,A -85,B 0,C 180,E1 -1389.359,E2 -1389.359} C_VEL
LIN {X 0,Y 587.355,Z 230.322,A -85,B 0,C 180,E1 -1392.112,E2 -1392.112} C_VEL
LIN {X 0,Y 587.304,Z 230.331,A -85,B 0,C 180,E1 -1395.089,E2 -1395.089} C_VEL
LIN {X 0,Y 587.341,Z 230.325,A -85,B 0,C 180,E1 -1397.928,E2 -1397.928} C_VEL
LIN {X 0,Y 587.326,Z 230.328,A -85,B 0,C 180,E1 -1401.058,E2 -1401.058} C_VEL
LIN {X 0,Y 587.342,Z 230.325,A -85,B 0,C 180,E1 -1403.292,E2 -1403.292} C_VEL
LIN {X 0,Y 587.354,Z 230.324,A -85,B 0,C 180,E1 -1405.781,E2 -1405.781} C_VEL
LIN {X 0,Y 587.345,Z 230.325,A -85,B 0,C 180,E1 -1408.233,E2 -1408.233} C_VEL
LIN {X 0,Y 587.34,Z 230.328,A -85,B 0,C 180,E1 -1410.867,E2 -1410.867} C_VEL
LIN {X 0,Y 587.355,Z 230.322,A -85,B 0,C 180,E1 -1413.818,E2 -1413.818} C_VEL
LIN {X 0,Y 587.316,Z 230.33,A -85,B 0,C 180,E1 -1416.742,E2 -1416.742} C_VEL
LIN {X 0,Y 587.328,Z 230.326,A -85,B 0,C 180,E1 -1419.696,E2 -1419.696} C_VEL
LIN {X 0,Y 587.351,Z 230.324,A -85,B 0,C 180,E1 -1422.595,E2 -1422.595} C_VEL
LIN {X 0,Y 587.356,Z 230.322,A -85,B 0,C 180,E1 -1425.74,E2 -1425.74} C_VEL
LIN {X 0,Y 587.354,Z 230.326,A -85,B 0,C 180,E1 -1428.859,E2 -1428.859} C_VEL
LIN {X 0,Y 587.367,Z 230.321,A -85,B 0,C 180,E1 -1431.746,E2 -1431.746} C_VEL
LIN {X 0,Y 587.353,Z 230.324,A -85,B 0,C 180,E1 -1434.508,E2 -1434.508} C_VEL
LIN {X 0,Y 587.375,Z 230.323,A -85,B 0,C 180,E1 -1437.258,E2 -1437.258} C_VEL
LIN {X 0,Y 587.371,Z 230.321,A -85,B 0,C 180,E1 -1440.001,E2 -1440.001} C_VEL
LIN {X 0,Y 587.362,Z 230.322,A -85,B 0,C 180,E1 -1442.744,E2 -1442.744} C_VEL
LIN {X 0,Y 587.353,Z 230.325,A -85,B 0,C 180,E1 -1445.494,E2 -1445.494} C_VEL
LIN {X 0,Y 587.361,Z 230.323,A -85,B 0,C 180,E1 -1448.256,E2 -1448.256} C_VEL
LIN {X 0,Y 587.341,Z 230.324,A -85,B 0,C 180,E1 -1451.135,E2 -1451.135} C_VEL
LIN {X 0,Y 587.36,Z 230.323,A -85,B 0,C 180,E1 -1454.262,E2 -1454.262} C_VEL
LIN {X 0,Y 587.347,Z 230.325,A -85,B 0,C 180,E1 -1457.407,E2 -1457.407} C_VEL
LIN {X 0,Y 587.324,Z 230.327,A -85,B 0,C 180,E1 -1460.306,E2 -1460.306} C_VEL
LIN {X 0,Y 587.318,Z 230.327,A -85,B 0,C 180,E1 -1463.26,E2 -1463.26} C_VEL
LIN {X 0,Y 587.329,Z 230.326,A -85,B 0,C 180,E1 -1465.518,E2 -1465.518} C_VEL
LIN {X 0,Y 587.347,Z 230.323,A -85,B 0,C 180,E1 -1467.818,E2 -1467.818} C_VEL
LIN {X 0,Y 587.328,Z 230.326,A -85,B 0,C 180,E1 -1470.51,E2 -1470.51} C_VEL
LIN {X 0,Y 587.334,Z 230.327,A -85,B 0,C 180,E1 -1473.112,E2 -1473.112} C_VEL
LIN {X 0,Y 587.301,Z 230.33,A -85,B 0,C 180,E1 -1475.9,E2 -1475.9} C_VEL
LIN {X 0,Y 587.333,Z 230.325,A -85,B 0,C 180,E1 -1478.48,E2 -1478.48} C_VEL
LIN {X 0,Y 587.335,Z 230.325,A -85,B 0,C 180,E1 -1481.158,E2 -1481.158} C_VEL
LIN {X 0,Y 587.325,Z 230.329,A -85,B 0,C 180,E1 -1484.114,E2 -1484.114} C_VEL
LIN {X 0,Y 587.316,Z 230.327,A -85,B 0,C 180,E1 -1486.995,E2 -1486.995} C_VEL
LIN {X 0,Y 587.317,Z 230.328,A -85,B 0,C 180,E1 -1489.747,E2 -1489.747} C_VEL
LIN {X 0,Y 587.342,Z 230.328,A -85,B 0,C 180,E1 -1492.393,E2 -1492.393} C_VEL
LIN {X 0,Y 587.354,Z 230.418,A -85,B 0,C 180,E1 -1493.999,E2 -1493.999} C_VEL
LIN {X 0,Y 587.506,Z 235.087,A -85,B 0,C 180,E1 -1495.79,E2 -1495.79} C_VEL
LIN {X 0,Y 587.469,Z 241.703,A -85,B 0,C 180,E1 -1498.239,E2 -1498.239} C_VEL
LIN {X 0,Y 587.364,Z 249.016,A -85,B 0,C 180,E1 -1500.865,E2 -1500.865} C_VEL
LIN {X 0,Y 587.315,Z 256.219,A -85,B 0,C 180,E1 -1503.338,E2 -1503.338} C_VEL
LIN {X 0,Y 587.341,Z 264.11,A -85,B 0,C 180,E1 -1505.994,E2 -1505.994} C_VEL
LIN {X 0,Y 587.298,Z 273.046,A -85,B 0,C 180,E1 -1508.972,E2 -1508.972} C_VEL
LIN {X 0,Y 587.267,Z 281.918,A -85,B 0,C 180,E1 -1511.872,E2 -1511.872} C_VEL
LIN {X 0,Y 587.247,Z 289.71,A -85,B 0,C 180,E1 -1514.379,E2 -1514.379} C_VEL
LIN {X 0,Y 587.207,Z 298.614,A -85,B 0,C 180,E1 -1517.208,E2 -1517.208} C_VEL
LIN {X 0,Y 587.18,Z 300.492,A -85,B 0,C 180,E1 -1517.8,E2 -1517.8} C_VEL
LIN {X 0,Y 587.752,Z 305.237,A -85,B 0,C 180,E1 -1517.9,E2 -1517.9} C_VEL
LIN {X 0,Y 587.68,Z 318.502,A -85,B 0,C 180,E1 -1518.226,E2 -1518.226} C_VEL
LIN {X 0,Y 587.568,Z 330.392,A -85,B 0,C 180,E1 -1518.656,E2 -1518.656} C_VEL
LIN {X 0,Y 587.492,Z 342.213,A -85,B 0,C 180,E1 -1519.227,E2 -1519.227} C_VEL
LIN {X 0,Y 587.467,Z 353.48,A -85,B 0,C 180,E1 -1519.924,E2 -1519.924} C_VEL
LIN {X 0,Y 587.384,Z 363.648,A -85,B 0,C 180,E1 -1520.705,E2 -1520.705} C_VEL
LIN {X 0,Y 587.34,Z 372.788,A -85,B 0,C 180,E1 -1521.571,E2 -1521.571} C_VEL
LIN {X 0,Y 587.259,Z 381.691,A -85,B 0,C 180,E1 -1522.608,E2 -1522.608} C_VEL
LIN {X 0,Y 587.195,Z 388.748,A -85,B 0,C 180,E1 -1523.627,E2 -1523.627} C_VEL
LIN {X 0,Y 587.211,Z 393.68,A -85,B 0,C 180,E1 -1524.506,E2 -1524.506} C_VEL
LIN {X 0,Y 587.189,Z 398.371,A -85,B 0,C 180,E1 -1525.538,E2 -1525.538} C_VEL
LIN {X 0,Y 587.193,Z 401.957,A -85,B 0,C 180,E1 -1526.569,E2 -1526.569} C_VEL
LIN {X 0,Y 587.132,Z 403.808,A -85,B 0,C 180,E1 -1527.256,E2 -1527.256} C_VEL
LIN {X 0,Y 587.141,Z 405.2,A -85,B 0,C 180,E1 -1527.942,E2 -1527.942} C_VEL
LIN {X 0,Y 587.14,Z 406.784,A -85,B 0,C 180,E1 -1529.314,E2 -1529.314} C_VEL
LIN {X 0,Y 587.137,Z 407,A -85,B 0,C 180,E1 -1530,E2 -1530} C_VEL
LIN {X 0,Y 587.147,Z 406.185,A -85,B 0,C 180,E1 -1531.372,E2 -1531.372} C_VEL
LIN {X 0,Y 587.141,Z 405.201,A -85,B 0,C 180,E1 -1532.058,E2 -1532.058} C_VEL
LIN {X 0,Y 587.132,Z 403.81,A -85,B 0,C 180,E1 -1532.744,E2 -1532.744} C_VEL
LIN {X 0,Y 587.213,Z 400.897,A -85,B 0,C 180,E1 -1533.774,E2 -1533.774} C_VEL
LIN {X 0,Y 587.147,Z 396.95,A -85,B 0,C 180,E1 -1534.806,E2 -1534.806} C_VEL
LIN {X 0,Y 587.218,Z 390.879,A -85,B 0,C 180,E1 -1536.011,E2 -1536.011} C_VEL
LIN {X 0,Y 587.245,Z 384.238,A -85,B 0,C 180,E1 -1537.046,E2 -1537.046} C_VEL
LIN {X 0,Y 587.299,Z 375.992,A -85,B 0,C 180,E1 -1538.083,E2 -1538.083} C_VEL
LIN {X 0,Y 587.343,Z 367.541,A -85,B 0,C 180,E1 -1538.949,E2 -1538.949} C_VEL
LIN {X 0,Y 587.421,Z 357.099,A -85,B 0,C 180,E1 -1539.816,E2 -1539.816} C_VEL
LIN {X 0,Y 587.475,Z 346.763,A -85,B 0,C 180,E1 -1540.511,E2 -1540.511} C_VEL
LIN {X 0,Y 587.53,Z 335.164,A -85,B 0,C 180,E1 -1541.133,E2 -1541.133} C_VEL
LIN {X 0,Y 587.623,Z 322.701,A -85,B 0,C 180,E1 -1541.636,E2 -1541.636} C_VEL
LIN {X 0,Y 587.732,Z 309.45,A -85,B 0,C 180,E1 -1542.013,E2 -1542.013} C_VEL
LIN {X 0,Y 587.533,Z 302.668,A -85,B 0,C 180,E1 -1542.154,E2 -1542.154} C_VEL
LIN {X 0,Y 587.179,Z 300.423,A -85,B 0,C 180,E1 -1542.222,E2 -1542.222} C_VEL
LIN {X 0,Y 587.219,Z 291.936,A -85,B 0,C 180,E1 -1544.911,E2 -1544.911} C_VEL
LIN {X 0,Y 587.283,Z 283.032,A -85,B 0,C 180,E1 -1547.767,E2 -1547.767} C_VEL
LIN {X 0,Y 587.292,Z 274.143,A -85,B 0,C 180,E1 -1550.666,E2 -1550.666} C_VEL
LIN {X 0,Y 587.339,Z 265.223,A -85,B 0,C 180,E1 -1553.631,E2 -1553.631} C_VEL
LIN {X 0,Y 587.307,Z 257.316,A -85,B 0,C 180,E1 -1556.279,E2 -1556.279} C_VEL
LIN {X 0,Y 587.353,Z 250.508,A -85,B 0,C 180,E1 -1558.595,E2 -1558.595} C_VEL
LIN {X 0,Y 587.449,Z 243.871,A -85,B 0,C 180,E1 -1560.959,E2 -1560.959} C_VEL
LIN {X 0,Y 587.495,Z 236.133,A -85,B 0,C 180,E1 -1563.797,E2 -1563.797} C_VEL
LIN {X 0,Y 587.422,Z 230.695,A -85,B 0,C 180,E1 -1565.89,E2 -1565.89} C_VEL
LIN {X 0,Y 587.347,Z 230.327,A -85,B 0,C 180,E1 -1566.107,E2 -1566.107} C_VEL
LIN {X 0,Y 587.322,Z 230.328,A -85,B 0,C 180,E1 -1568.94,E2 -1568.94} C_VEL
LIN {X 0,Y 587.352,Z 230.325,A -85,B 0,C 180,E1 -1572.071,E2 -1572.071} C_VEL
LIN {X 0,Y 587.314,Z 230.329,A -85,B 0,C 180,E1 -1575.088,E2 -1575.088} C_VEL
LIN {X 0,Y 587.35,Z 230.324,A -85,B 0,C 180,E1 -1577.927,E2 -1577.927} C_VEL
LIN {X 0,Y 587.332,Z 230.326,A -85,B 0,C 180,E1 -1581.057,E2 -1581.057} C_VEL
LIN {X 0,Y 587.352,Z 230.324,A -85,B 0,C 180,E1 -1583.29,E2 -1583.29} C_VEL
LIN {X 0,Y 587.364,Z 230.324,A -85,B 0,C 180,E1 -1585.78,E2 -1585.78} C_VEL
LIN {X 0,Y 587.351,Z 230.324,A -85,B 0,C 180,E1 -1588.231,E2 -1588.231} C_VEL
LIN {X 0,Y 587.345,Z 230.327,A -85,B 0,C 180,E1 -1590.865,E2 -1590.865} C_VEL
LIN {X 0,Y 587.353,Z 230.325,A -85,B 0,C 180,E1 -1593.818,E2 -1593.818} C_VEL
LIN {X 0,Y 587.334,Z 230.329,A -85,B 0,C 180,E1 -1595.993,E2 -1595.993} C_VEL
LIN {X 0,Y 587.318,Z 230.329,A -85,B 0,C 180,E1 -1598.225,E2 -1598.225} C_VEL
LIN {X 0,Y 587.345,Z 230.327,A -85,B 0,C 180,E1 -1601.15,E2 -1601.15} C_VEL
LIN {X 0,Y 587.344,Z 230.326,A -85,B 0,C 180,E1 -1603.31,E2 -1603.31} C_VEL
LIN {X 0,Y 587.357,Z 230.325,A -85,B 0,C 180,E1 -1606.154,E2 -1606.154} C_VEL
LIN {X 0,Y 587.34,Z 230.326,A -85,B 0,C 180,E1 -1608.962,E2 -1608.962} C_VEL
LIN {X 0,Y 587.367,Z 230.322,A -85,B 0,C 180,E1 -1611.744,E2 -1611.744} C_VEL
LIN {X 0,Y 587.356,Z 230.325,A -85,B 0,C 180,E1 -1614.506,E2 -1614.506} C_VEL
LIN {X 0,Y 587.374,Z 230.322,A -85,B 0,C 180,E1 -1617.256,E2 -1617.256} C_VEL
LIN {X 0,Y 587.374,Z 230.321,A -85,B 0,C 180,E1 -1619.999,E2 -1619.999} C_VEL
LIN {X 0,Y 587.376,Z 230.323,A -85,B 0,C 180,E1 -1622.742,E2 -1622.742} C_VEL
LIN {X 0,Y 587.351,Z 230.325,A -85,B 0,C 180,E1 -1625.492,E2 -1625.492} C_VEL
LIN {X 0,Y 587.368,Z 230.322,A -85,B 0,C 180,E1 -1628.254,E2 -1628.254} C_VEL
LIN {X 0,Y 587.326,Z 230.328,A -85,B 0,C 180,E1 -1630.339,E2 -1630.339} C_VEL
LIN {X 0,Y 587.336,Z 230.983,A -85,B 0,C 180,E1 -1631.133,E2 -1631.133} C_VEL
LIN {X 0,Y 587.307,Z 236.283,A -85,B 0,C 180,E1 -1634.242,E2 -1634.242} C_VEL
LIN {X 0,Y 587.282,Z 241.784,A -85,B 0,C 180,E1 -1637.407,E2 -1637.407} C_VEL
LIN {X 0,Y 587.261,Z 243.193,A -85,B 0,C 180,E1 -1638.198,E2 -1638.198} C_VEL
LIN {X 0,Y 586.592,Z 244.27,A -85,B 0,C 180,E1 -1638.76,E2 -1638.76} C_VEL
LIN {X 0,Y 583.77,Z 246.145,A -85,B 0,C 180,E1 -1639.67,E2 -1639.67} C_VEL
LIN {X 0,Y 581.363,Z 247.646,A -85,B 0,C 180,E1 -1640.403,E2 -1640.403} C_VEL
LIN {X 0,Y 580.287,Z 248.719,A -85,B 0,C 180,E1 -1640.969,E2 -1640.969} C_VEL
LIN {X 0,Y 580.176,Z 249.058,A -85,B 0,C 180,E1 -1641.161,E2 -1641.161} C_VEL
LIN {X 0,Y 580.126,Z 253.256,A -85,B 0,C 180,E1 -1643.563,E2 -1643.563} C_VEL
LIN {X 0,Y 580.075,Z 258.968,A -85,B 0,C 180,E1 -1646.632,E2 -1646.632} C_VEL
LIN {X 0,Y 580.074,Z 263.965,A -85,B 0,C 180,E1 -1649.272,E2 -1649.272} C_VEL
LIN {X 0,Y 580.043,Z 269.189,A -85,B 0,C 180,E1 -1651.992,E2 -1651.992} C_VEL
LIN {X 0,Y 580.104,Z 272.552,A -85,B 0,C 180,E1 -1653.727,E2 -1653.727} C_VEL
LIN {X 0,Y 580.801,Z 278.915,A -85,B 0,C 180,E1 -1653.873,E2 -1653.873} C_VEL
LIN {X 0,Y 580.662,Z 292.155,A -85,B 0,C 180,E1 -1654.249,E2 -1654.249} C_VEL
LIN {X 0,Y 580.556,Z 304.141,A -85,B 0,C 180,E1 -1654.729,E2 -1654.729} C_VEL
LIN {X 0,Y 580.517,Z 315.274,A -85,B 0,C 180,E1 -1655.314,E2 -1655.314} C_VEL
LIN {X 0,Y 580.408,Z 326.426,A -85,B 0,C 180,E1 -1656.058,E2 -1656.058} C_VEL
LIN {X 0,Y 580.307,Z 336.993,A -85,B 0,C 180,E1 -1656.937,E2 -1656.937} C_VEL
LIN {X 0,Y 580.26,Z 346.176,A -85,B 0,C 180,E1 -1657.885,E2 -1657.885} C_VEL
LIN {X 0,Y 580.168,Z 353.578,A -85,B 0,C 180,E1 -1658.819,E2 -1658.819} C_VEL
LIN {X 0,Y 580.122,Z 360.793,A -85,B 0,C 180,E1 -1659.945,E2 -1659.945} C_VEL
LIN {X 0,Y 580.094,Z 365.493,A -85,B 0,C 180,E1 -1660.859,E2 -1660.859} C_VEL
LIN {X 0,Y 580.096,Z 369.346,A -85,B 0,C 180,E1 -1661.783,E2 -1661.783} C_VEL
LIN {X 0,Y 580.069,Z 372.416,A -85,B 0,C 180,E1 -1662.724,E2 -1662.724} C_VEL
LIN {X 0,Y 580.018,Z 374.678,A -85,B 0,C 180,E1 -1663.681,E2 -1663.681} C_VEL
LIN {X 0,Y 580.066,Z 376.172,A -85,B 0,C 180,E1 -1664.644,E2 -1664.644} C_VEL
LIN {X 0,Y 580.057,Z 376.912,A -85,B 0,C 180,E1 -1665.629,E2 -1665.629} C_VEL
LIN {X 0,Y 580.021,Z 376.855,A -85,B 0,C 180,E1 -1666.634,E2 -1666.634} C_VEL
LIN {X 0,Y 580.051,Z 375.935,A -85,B 0,C 180,E1 -1667.652,E2 -1667.652} C_VEL
LIN {X 0,Y 580.033,Z 374.086,A -85,B 0,C 180,E1 -1668.695,E2 -1668.695} C_VEL
LIN {X 0,Y 580.089,Z 370.254,A -85,B 0,C 180,E1 -1670.051,E2 -1670.051} C_VEL
LIN {X 0,Y 580.117,Z 365.745,A -85,B 0,C 180,E1 -1671.176,E2 -1671.176} C_VEL
LIN {X 0,Y 580.105,Z 359.707,A -85,B 0,C 180,E1 -1672.332,E2 -1672.332} C_VEL
LIN {X 0,Y 580.184,Z 353.099,A -85,B 0,C 180,E1 -1673.338,E2 -1673.338} C_VEL
LIN {X 0,Y 580.248,Z 345.868,A -85,B 0,C 180,E1 -1674.241,E2 -1674.241} C_VEL
LIN {X 0,Y 580.314,Z 336.465,A -85,B 0,C 180,E1 -1675.201,E2 -1675.201} C_VEL
LIN {X 0,Y 580.39,Z 326.231,A -85,B 0,C 180,E1 -1676.047,E2 -1676.047} C_VEL
LIN {X 0,Y 580.412,Z 315.989,A -85,B 0,C 180,E1 -1676.733,E2 -1676.733} C_VEL
LIN {X 0,Y 580.518,Z 304.355,A -85,B 0,C 180,E1 -1677.352,E2 -1677.352} C_VEL
LIN {X 0,Y 580.648,Z 292.726,A -85,B 0,C 180,E1 -1677.822,E2 -1677.822} C_VEL
LIN {X 0,Y 580.755,Z 279.54,A -85,B 0,C 180,E1 -1678.202,E2 -1678.202} C_VEL
LIN {X 0,Y 580.422,Z 275.006,A -85,B 0,C 180,E1 -1678.305,E2 -1678.305} C_VEL
LIN {X 0,Y 580.044,Z 272.534,A -85,B 0,C 180,E1 -1678.373,E2 -1678.373} C_VEL
LIN {X 0,Y 580.068,Z 267.425,A -85,B 0,C 180,E1 -1681.012,E2 -1681.012} C_VEL
LIN {X 0,Y 580.042,Z 261.456,A -85,B 0,C 180,E1 -1684.14,E2 -1684.14} C_VEL
LIN {X 0,Y 580.093,Z 257.137,A -85,B 0,C 180,E1 -1686.435,E2 -1686.435} C_VEL
LIN {X 0,Y 580.127,Z 251.62,A -85,B 0,C 180,E1 -1689.432,E2 -1689.432} C_VEL
LIN {X 0,Y 580.128,Z 247.754,A -85,B 0,C 180,E1 -1691.641,E2 -1691.641} C_VEL
LIN {X 0,Y 580.182,Z 243.904,A -85,B 0,C 180,E1 -1693.823,E2 -1693.823} C_VEL
LIN {X 0,Y 580.191,Z 238.921,A -85,B 0,C 180,E1 -1696.694,E2 -1696.694} C_VEL
LIN {X 0,Y 580.263,Z 234.081,A -85,B 0,C 180,E1 -1699.533,E2 -1699.533} C_VEL
LIN {X 0,Y 580.228,Z 231.748,A -85,B 0,C 180,E1 -1700.941,E2 -1700.941} C_VEL
LIN {X 0,Y 580.261,Z 231.204,A -85,B 0,C 180,E1 -1701.643,E2 -1701.643} C_VEL
LIN {X 0,Y 580.272,Z 231.207,A -85,B 0,C 180,E1 -1703.742,E2 -1703.742} C_VEL
LIN {X 0,Y 580.269,Z 231.207,A -85,B 0,C 180,E1 -1705.833,E2 -1705.833} C_VEL
LIN {X 0,Y 580.324,Z 231.198,A -85,B 0,C 180,E1 -1707.918,E2 -1707.918} C_VEL
LIN {X 0,Y 580.358,Z 231.197,A -85,B 0,C 180,E1 -1710.694,E2 -1710.694} C_VEL
LIN {X 0,Y 580.282,Z 231.205,A -85,B 0,C 180,E1 -1713.472,E2 -1713.472} C_VEL
LIN {X 0,Y 580.318,Z 231.202,A -85,B 0,C 180,E1 -1715.56,E2 -1715.56} C_VEL
LIN {X 0,Y 580.328,Z 231.198,A -85,B 0,C 180,E1 -1718.356,E2 -1718.356} C_VEL
LIN {X 0,Y 580.323,Z 231.199,A -85,B 0,C 180,E1 -1721.208,E2 -1721.208} C_VEL
LIN {X 0,Y 580.305,Z 231.201,A -85,B 0,C 180,E1 -1724.339,E2 -1724.339} C_VEL
LIN {X 0,Y 580.306,Z 231.2,A -85,B 0,C 180,E1 -1726.916,E2 -1726.916} C_VEL
LIN {X 0,Y 580.298,Z 231.203,A -85,B 0,C 180,E1 -1729.822,E2 -1729.822} C_VEL
LIN {X 0,Y 580.319,Z 231.199,A -85,B 0,C 180,E1 -1732.801,E2 -1732.801} C_VEL
LIN {X 0,Y 580.295,Z 231.203,A -85,B 0,C 180,E1 -1735.08,E2 -1735.08} C_VEL
LIN {X 0,Y 580.31,Z 231.2,A -85,B 0,C 180,E1 -1737.864,E2 -1737.864} C_VEL
LIN {X 0,Y 580.289,Z 231.205,A -85,B 0,C 180,E1 -1740.698,E2 -1740.698} C_VEL
LIN {X 0,Y 580.294,Z 231.205,A -85,B 0,C 180,E1 -1743.317,E2 -1743.317} C_VEL
LIN {X 0,Y 580.316,Z 231.201,A -85,B 0,C 180,E1 -1745.768,E2 -1745.768} C_VEL
LIN {X 0,Y 580.28,Z 231.206,A -85,B 0,C 180,E1 -1748.146,E2 -1748.146} C_VEL
LIN {X 0,Y 580.293,Z 231.202,A -85,B 0,C 180,E1 -1750.843,E2 -1750.843} C_VEL
LIN {X 0,Y 580.279,Z 231.205,A -85,B 0,C 180,E1 -1753.657,E2 -1753.657} C_VEL
LIN {X 0,Y 580.279,Z 231.206,A -85,B 0,C 180,E1 -1756.608,E2 -1756.608} C_VEL
LIN {X 0,Y 580.292,Z 231.203,A -85,B 0,C 180,E1 -1759.158,E2 -1759.158} C_VEL
LIN {X 0,Y 580.28,Z 231.204,A -85,B 0,C 180,E1 -1761.927,E2 -1761.927} C_VEL
LIN {X 0,Y 580.296,Z 231.202,A -85,B 0,C 180,E1 -1764.457,E2 -1764.457} C_VEL
LIN {X 0,Y 580.281,Z 231.205,A -85,B 0,C 180,E1 -1766.976,E2 -1766.976} C_VEL
LIN {X 0,Y 580.299,Z 231.203,A -85,B 0,C 180,E1 -1769.427,E2 -1769.427} C_VEL
LIN {X 0,Y 580.308,Z 231.203,A -85,B 0,C 180,E1 -1772.138,E2 -1772.138} C_VEL
LIN {X 0,Y 580.301,Z 231.201,A -85,B 0,C 180,E1 -1774.921,E2 -1774.921} C_VEL
LIN {X 0,Y 580.264,Z 231.209,A -85,B 0,C 180,E1 -1777.948,E2 -1777.948} C_VEL
LIN {X 0,Y 580.308,Z 231.2,A -85,B 0,C 180,E1 -1780.915,E2 -1780.915} C_VEL
LIN {X 0,Y 580.274,Z 231.206,A -85,B 0,C 180,E1 -1783.826,E2 -1783.826} C_VEL
LIN {X 0,Y 580.317,Z 231.199,A -85,B 0,C 180,E1 -1785.984,E2 -1785.984} C_VEL
LIN {X 0,Y 580.323,Z 231.202,A -85,B 0,C 180,E1 -1788.828,E2 -1788.828} C_VEL
LIN {X 0,Y 580.33,Z 231.198,A -85,B 0,C 180,E1 -1791.645,E2 -1791.645} C_VEL
LIN {X 0,Y 580.318,Z 231.2,A -85,B 0,C 180,E1 -1794.441,E2 -1794.441} C_VEL
LIN {X 0,Y 580.34,Z 231.199,A -85,B 0,C 180,E1 -1797.224,E2 -1797.224} C_VEL
LIN {X 0,Y 580.34,Z 231.197,A -85,B 0,C 180,E1 -1800.001,E2 -1800.001} C_VEL
LIN {X 0,Y 580.33,Z 231.198,A -85,B 0,C 180,E1 -1802.777,E2 -1802.777} C_VEL
LIN {X 0,Y 580.319,Z 231.202,A -85,B 0,C 180,E1 -1805.561,E2 -1805.561} C_VEL
LIN {X 0,Y 580.323,Z 231.199,A -85,B 0,C 180,E1 -1808.357,E2 -1808.357} C_VEL
LIN {X 0,Y 580.293,Z 231.202,A -85,B 0,C 180,E1 -1811.192,E2 -1811.192} C_VEL
LIN {X 0,Y 580.323,Z 231.202,A -85,B 0,C 180,E1 -1814.018,E2 -1814.018} C_VEL
LIN {X 0,Y 580.308,Z 231.2,A -85,B 0,C 180,E1 -1816.915,E2 -1816.915} C_VEL
LIN {X 0,Y 580.301,Z 231.203,A -85,B 0,C 180,E1 -1819.823,E2 -1819.823} C_VEL
LIN {X 0,Y 580.293,Z 231.203,A -85,B 0,C 180,E1 -1822.803,E2 -1822.803} C_VEL
LIN {X 0,Y 580.302,Z 231.202,A -85,B 0,C 180,E1 -1825.081,E2 -1825.081} C_VEL
LIN {X 0,Y 580.301,Z 231.203,A -85,B 0,C 180,E1 -1828.186,E2 -1828.186} C_VEL
LIN {X 0,Y 580.281,Z 231.206,A -85,B 0,C 180,E1 -1830.696,E2 -1830.696} C_VEL
LIN {X 0,Y 580.28,Z 231.207,A -85,B 0,C 180,E1 -1833.314,E2 -1833.314} C_VEL
LIN {X 0,Y 580.27,Z 231.207,A -85,B 0,C 180,E1 -1835.761,E2 -1835.761} C_VEL
LIN {X 0,Y 580.288,Z 231.205,A -85,B 0,C 180,E1 -1838.147,E2 -1838.147} C_VEL
LIN {X 0,Y 580.298,Z 231.202,A -85,B 0,C 180,E1 -1840.844,E2 -1840.844} C_VEL
LIN {X 0,Y 580.277,Z 231.205,A -85,B 0,C 180,E1 -1843.659,E2 -1843.659} C_VEL
LIN {X 0,Y 580.275,Z 231.206,A -85,B 0,C 180,E1 -1846.61,E2 -1846.61} C_VEL
LIN {X 0,Y 580.299,Z 231.202,A -85,B 0,C 180,E1 -1849.157,E2 -1849.157} C_VEL
LIN {X 0,Y 580.287,Z 231.203,A -85,B 0,C 180,E1 -1851.928,E2 -1851.928} C_VEL
LIN {X 0,Y 580.286,Z 231.337,A -85,B 0,C 180,E1 -1853.853,E2 -1853.853} C_VEL
LIN {X 0,Y 580.551,Z 233.969,A -85,B 0,C 180,E1 -1854.899,E2 -1854.899} C_VEL
LIN {X 0,Y 580.491,Z 240.576,A -85,B 0,C 180,E1 -1857.401,E2 -1857.401} C_VEL
LIN {X 0,Y 580.406,Z 248.304,A -85,B 0,C 180,E1 -1860.234,E2 -1860.234} C_VEL
LIN {X 0,Y 580.294,Z 256.105,A -85,B 0,C 180,E1 -1862.989,E2 -1862.989} C_VEL
LIN {X 0,Y 580.296,Z 264.068,A -85,B 0,C 180,E1 -1865.684,E2 -1865.684} C_VEL
LIN {X 0,Y 580.266,Z 273.014,A -85,B 0,C 180,E1 -1868.694,E2 -1868.694} C_VEL
LIN {X 0,Y 580.203,Z 281.918,A -85,B 0,C 180,E1 -1871.643,E2 -1871.643} C_VEL
LIN {X 0,Y 580.176,Z 290.823,A -85,B 0,C 180,E1 -1874.544,E2 -1874.544} C_VEL
LIN {X 0,Y 580.135,Z 299.727,A -85,B 0,C 180,E1 -1877.405,E2 -1877.405} C_VEL
LIN {X 0,Y 580.11,Z 300.492,A -85,B 0,C 180,E1 -1877.649,E2 -1877.649} C_VEL
LIN {X 0,Y 580.811,Z 306.377,A -85,B 0,C 180,E1 -1877.775,E2 -1877.775} C_VEL
LIN {X 0,Y 580.714,Z 318.503,A -85,B 0,C 180,E1 -1878.083,E2 -1878.083} C_VEL
LIN {X 0,Y 580.616,Z 330.32,A -85,B 0,C 180,E1 -1878.515,E2 -1878.515} C_VEL
LIN {X 0,Y 580.489,Z 342.212,A -85,B 0,C 180,E1 -1879.096,E2 -1879.096} C_VEL
LIN {X 0,Y 580.456,Z 353.482,A -85,B 0,C 180,E1 -1879.801,E2 -1879.801} C_VEL
LIN {X 0,Y 580.352,Z 363.648,A -85,B 0,C 180,E1 -1880.591,E2 -1880.591} C_VEL
LIN {X 0,Y 580.279,Z 372.787,A -85,B 0,C 180,E1 -1881.468,E2 -1881.468} C_VEL
LIN {X 0,Y 580.199,Z 381.69,A -85,B 0,C 180,E1 -1882.518,E2 -1882.518} C_VEL
LIN {X 0,Y 580.12,Z 388.467,A -85,B 0,C 180,E1 -1883.505,E2 -1883.505} C_VEL
LIN {X 0,Y 580.139,Z 393.68,A -85,B 0,C 180,E1 -1884.438,E2 -1884.438} C_VEL
LIN {X 0,Y 580.108,Z 398.372,A -85,B 0,C 180,E1 -1885.483,E2 -1885.483} C_VEL
LIN {X 0,Y 580.123,Z 401.957,A -85,B 0,C 180,E1 -1886.527,E2 -1886.527} C_VEL
LIN {X 0,Y 580.043,Z 403.808,A -85,B 0,C 180,E1 -1887.222,E2 -1887.222} C_VEL
LIN {X 0,Y 580.04,Z 405.199,A -85,B 0,C 180,E1 -1887.917,E2 -1887.917} C_VEL
LIN {X 0,Y 580.04,Z 406.785,A -85,B 0,C 180,E1 -1889.306,E2 -1889.306} C_VEL
LIN {X 0,Y 580.037,Z 407,A -85,B 0,C 180,E1 -1890,E2 -1890} C_VEL
LIN {X 0,Y 580.047,Z 406.186,A -85,B 0,C 180,E1 -1891.388,E2 -1891.388} C_VEL
LIN {X 0,Y 580.04,Z 405.2,A -85,B 0,C 180,E1 -1892.083,E2 -1892.083} C_VEL
LIN {X 0,Y 580.043,Z 403.81,A -85,B 0,C 180,E1 -1892.778,E2 -1892.778} C_VEL
LIN {X 0,Y 580.11,Z 400.896,A -85,B 0,C 180,E1 -1893.82,E2 -1893.82} C_VEL
LIN {X 0,Y 580.053,Z 396.95,A -85,B 0,C 180,E1 -1894.865,E2 -1894.865} C_VEL
LIN {X 0,Y 580.139,Z 390.878,A -85,B 0,C 180,E1 -1896.085,E2 -1896.085} C_VEL
LIN {X 0,Y 580.184,Z 384.239,A -85,B 0,C 180,E1 -1897.132,E2 -1897.132} C_VEL
LIN {X 0,Y 580.25,Z 375.993,A -85,B 0,C 180,E1 -1898.182,E2 -1898.182} C_VEL
LIN {X 0,Y 580.308,Z 367.541,A -85,B 0,C 180,E1 -1899.058,E2 -1899.058} C_VEL
LIN {X 0,Y 580.423,Z 357.101,A -85,B 0,C 180,E1 -1899.936,E2 -1899.936} C_VEL
LIN {X 0,Y 580.477,Z 346.761,A -85,B 0,C 180,E1 -1900.64,E2 -1900.64} C_VEL
LIN {X 0,Y 580.563,Z 335.596,A -85,B 0,C 180,E1 -1901.247,E2 -1901.247} C_VEL
LIN {X 0,Y 580.65,Z 323.777,A -85,B 0,C 180,E1 -1901.741,E2 -1901.741} C_VEL
LIN {X 0,Y 580.782,Z 310.363,A -85,B 0,C 180,E1 -1902.137,E2 -1902.137} C_VEL
LIN {X 0,Y 580.682,Z 304.102,A -85,B 0,C 180,E1 -1902.272,E2 -1902.272} C_VEL
LIN {X 0,Y 580.11,Z 300.493,A -85,B 0,C 180,E1 -1902.351,E2 -1902.351} C_VEL
LIN {X 0,Y 580.156,Z 291.936,A -85,B 0,C 180,E1 -1905.096,E2 -1905.096} C_VEL
LIN {X 0,Y 580.21,Z 283.032,A -85,B 0,C 180,E1 -1907.991,E2 -1907.991} C_VEL
LIN {X 0,Y 580.237,Z 275.241,A -85,B 0,C 180,E1 -1910.564,E2 -1910.564} C_VEL
LIN {X 0,Y 580.261,Z 267.98,A -85,B 0,C 180,E1 -1913.001,E2 -1913.001} C_VEL
LIN {X 0,Y 580.322,Z 260.593,A -85,B 0,C 180,E1 -1915.462,E2 -1915.462} C_VEL
LIN {X 0,Y 580.332,Z 252.667,A -85,B 0,C 180,E1 -1918.183,E2 -1918.183} C_VEL
LIN {X 0,Y 580.436,Z 245.612,A -85,B 0,C 180,E1 -1920.719,E2 -1920.719} C_VEL
LIN {X 0,Y 580.517,Z 238.491,A -85,B 0,C 180,E1 -1923.348,E2 -1923.348} C_VEL
LIN {X 0,Y 580.487,Z 232.213,A -85,B 0,C 180,E1 -1925.789,E2 -1925.789} C_VEL
LIN {X 0,Y 580.318,Z 231.202,A -85,B 0,C 180,E1 -1926.231,E2 -1926.231} C_VEL
LIN {X 0,Y 580.295,Z 231.205,A -85,B 0,C 180,E1 -1929.184,E2 -1929.184} C_VEL
LIN {X 0,Y 580.313,Z 231.201,A -85,B 0,C 180,E1 -1931.765,E2 -1931.765} C_VEL
LIN {X 0,Y 580.267,Z 231.207,A -85,B 0,C 180,E1 -1934.625,E2 -1934.625} C_VEL
LIN {X 0,Y 580.283,Z 231.206,A -85,B 0,C 180,E1 -1937.627,E2 -1937.627} C_VEL
LIN {X 0,Y 580.291,Z 231.204,A -85,B 0,C 180,E1 -1940.066,E2 -1940.066} C_VEL
LIN {X 0,Y 580.299,Z 231.202,A -85,B 0,C 180,E1 -1943.064,E2 -1943.064} C_VEL
LIN {X 0,Y 580.301,Z 231.203,A -85,B 0,C 180,E1 -1945.439,E2 -1945.439} C_VEL
LIN {X 0,Y 580.306,Z 231.202,A -85,B 0,C 180,E1 -1947.967,E2 -1947.967} C_VEL
LIN {X 0,Y 580.3,Z 231.204,A -85,B 0,C 180,E1 -1950.689,E2 -1950.689} C_VEL
LIN {X 0,Y 580.276,Z 231.205,A -85,B 0,C 180,E1 -1953.376,E2 -1953.376} C_VEL
LIN {X 0,Y 580.296,Z 231.203,A -85,B 0,C 180,E1 -1955.683,E2 -1955.683} C_VEL
LIN {X 0,Y 580.269,Z 231.208,A -85,B 0,C 180,E1 -1957.947,E2 -1957.947} C_VEL
LIN {X 0,Y 580.312,Z 231.202,A -85,B 0,C 180,E1 -1960.913,E2 -1960.913} C_VEL
LIN {X 0,Y 580.276,Z 231.205,A -85,B 0,C 180,E1 -1963.825,E2 -1963.825} C_VEL
LIN {X 0,Y 580.322,Z 231.2,A -85,B 0,C 180,E1 -1965.982,E2 -1965.982} C_VEL
LIN {X 0,Y 580.324,Z 231.199,A -85,B 0,C 180,E1 -1968.827,E2 -1968.827} C_VEL
LIN {X 0,Y 580.33,Z 231.199,A -85,B 0,C 180,E1 -1971.643,E2 -1971.643} C_VEL
LIN {X 0,Y 580.321,Z 231.202,A -85,B 0,C 180,E1 -1974.439,E2 -1974.439} C_VEL
LIN {X 0,Y 580.339,Z 231.198,A -85,B 0,C 180,E1 -1977.223,E2 -1977.223} C_VEL
LIN {X 0,Y 580.344,Z 231.197,A -85,B 0,C 180,E1 -1979.999,E2 -1979.999} C_VEL
LIN {X 0,Y 580.341,Z 231.199,A -85,B 0,C 180,E1 -1982.776,E2 -1982.776} C_VEL
LIN {X 0,Y 580.318,Z 231.202,A -85,B 0,C 180,E1 -1985.559,E2 -1985.559} C_VEL
LIN {X 0,Y 580.331,Z 231.199,A -85,B 0,C 180,E1 -1988.355,E2 -1988.355} C_VEL
LIN {X 0,Y 580.285,Z 231.205,A -85,B 0,C 180,E1 -1990.466,E2 -1990.466} C_VEL
LIN {X 0,Y 580.288,Z 231.935,A -85,B 0,C 180,E1 -1991.19,E2 -1991.19} C_VEL
LIN {X 0,Y 580.268,Z 237.211,A -85,B 0,C 180,E1 -1994.324,E2 -1994.324} C_VEL
LIN {X 0,Y 580.216,Z 241.637,A -85,B 0,C 180,E1 -1996.899,E2 -1996.899} C_VEL
LIN {X 0,Y 580.178,Z 246.796,A -85,B 0,C 180,E1 -1999.826,E2 -1999.826} C_VEL
LIN {X 0,Y 580.176,Z 249.058,A -85,B 0,C 180,E1 -2001.161,E2 -2001.161} C_VEL
LIN {X 0,Y 579.444,Z 250.11,A -85,B 0,C 180,E1 -2001.731,E2 -2001.731} C_VEL
LIN {X 0,Y 576.555,Z 251.988,A -85,B 0,C 180,E1 -2002.654,E2 -2002.654} C_VEL
LIN {X 0,Y 574.146,Z 253.506,A -85,B 0,C 180,E1 -2003.396,E2 -2003.396} C_VEL
LIN {X 0,Y 573.109,Z 254.601,A -85,B 0,C 180,E1 -2003.97,E2 -2003.97} C_VEL
LIN {X 0,Y 573.02,Z 254.947,A -85,B 0,C 180,E1 -2004.165,E2 -2004.165} C_VEL
LIN {X 0,Y 573.007,Z 260.089,A -85,B 0,C 180,E1 -2006.987,E2 -2006.987} C_VEL
LIN {X 0,Y 572.975,Z 264.689,A -85,B 0,C 180,E1 -2009.442,E2 -2009.442} C_VEL
LIN {X 0,Y 572.955,Z 269.893,A -85,B 0,C 180,E1 -2012.183,E2 -2012.183} C_VEL
LIN {X 0,Y 573,Z 272.663,A -85,B 0,C 180,E1 -2013.578,E2 -2013.578} C_VEL
LIN {X 0,Y 573.85,Z 279.251,A -85,B 0,C 180,E1 -2013.732,E2 -2013.732} C_VEL
LIN {X 0,Y 573.716,Z 291.589,A -85,B 0,C 180,E1 -2014.085,E2 -2014.085} C_VEL
LIN {X 0,Y 573.609,Z 303.675,A -85,B 0,C 180,E1 -2014.569,E2 -2014.569} C_VEL
LIN {X 0,Y 573.505,Z 315.004,A -85,B 0,C 180,E1 -2015.165,E2 -2015.165} C_VEL
LIN {X 0,Y 573.408,Z 326.552,A -85,B 0,C 180,E1 -2015.945,E2 -2015.945} C_VEL
LIN {X 0,Y 573.295,Z 336.813,A -85,B 0,C 180,E1 -2016.808,E2 -2016.808} C_VEL
LIN {X 0,Y 573.223,Z 344.858,A -85,B 0,C 180,E1 -2017.633,E2 -2017.633} C_VEL
LIN {X 0,Y 573.095,Z 353.455,A -85,B 0,C 180,E1 -2018.712,E2 -2018.712} C_VEL
LIN {X 0,Y 573.066,Z 360.615,A -85,B 0,C 180,E1 -2019.839,E2 -2019.839} C_VEL
LIN {X 0,Y 573.011,Z 366.464,A -85,B 0,C 180,E1 -2021.007,E2 -2021.007} C_VEL
LIN {X 0,Y 573.002,Z 370.182,A -85,B 0,C 180,E1 -2021.968,E2 -2021.968} C_VEL
LIN {X 0,Y 572.97,Z 372.213,A -85,B 0,C 180,E1 -2022.613,E2 -2022.613} C_VEL
LIN {X 0,Y 572.919,Z 374.648,A -85,B 0,C 180,E1 -2023.636,E2 -2023.636} C_VEL
LIN {X 0,Y 572.966,Z 376.198,A -85,B 0,C 180,E1 -2024.65,E2 -2024.65} C_VEL
LIN {X 0,Y 572.956,Z 376.916,A -85,B 0,C 180,E1 -2025.64,E2 -2025.64} C_VEL
LIN {X 0,Y 572.923,Z 376.871,A -85,B 0,C 180,E1 -2026.612,E2 -2026.612} C_VEL
LIN {X 0,Y 572.973,Z 376.042,A -85,B 0,C 180,E1 -2027.576,E2 -2027.576} C_VEL
LIN {X 0,Y 572.961,Z 373.484,A -85,B 0,C 180,E1 -2028.988,E2 -2028.988} C_VEL
LIN {X 0,Y 573.002,Z 370.808,A -85,B 0,C 180,E1 -2029.941,E2 -2029.941} C_VEL
LIN {X 0,Y 573.02,Z 367.079,A -85,B 0,C 180,E1 -2030.938,E2 -2030.938} C_VEL
LIN {X 0,Y 573.045,Z 362.276,A -85,B 0,C 180,E1 -2031.949,E2 -2031.949} C_VEL
LIN {X 0,Y 573.085,Z 355.629,A -85,B 0,C 180,E1 -2033.066,E2 -2033.066} C_VEL
LIN {X 0,Y 573.183,Z 347.037,A -85,B 0,C 180,E1 -2034.204,E2 -2034.204} C_VEL
LIN {X 0,Y 573.262,Z 337.464,A -85,B 0,C 180,E1 -2035.223,E2 -2035.223} C_VEL
LIN {X 0,Y 573.369,Z 327.179,A -85,B 0,C 180,E1 -2036.098,E2 -2036.098} C_VEL
LIN {X 0,Y 573.416,Z 316.338,A -85,B 0,C 180,E1 -2036.843,E2 -2036.843} C_VEL
LIN {X 0,Y 573.556,Z 304.676,A -85,B 0,C 180,E1 -2037.476,E2 -2037.476} C_VEL
LIN {X 0,Y 573.707,Z 292.298,A -85,B 0,C 180,E1 -2037.981,E2 -2037.981} C_VEL
LIN {X 0,Y 573.825,Z 279.059,A -85,B 0,C 180,E1 -2038.363,E2 -2038.363} C_VEL
LIN {X 0,Y 572.928,Z 272.538,A -85,B 0,C 180,E1 -2038.527,E2 -2038.527} C_VEL
LIN {X 0,Y 572.966,Z 267.009,A -85,B 0,C 180,E1 -2041.421,E2 -2041.421} C_VEL
LIN {X 0,Y 572.985,Z 262.528,A -85,B 0,C 180,E1 -2043.797,E2 -2043.797} C_VEL
LIN {X 0,Y 573.026,Z 256.762,A -85,B 0,C 180,E1 -2046.901,E2 -2046.901} C_VEL
LIN {X 0,Y 573.065,Z 251.423,A -85,B 0,C 180,E1 -2049.917,E2 -2049.917} C_VEL
LIN {X 0,Y 573.069,Z 247.542,A -85,B 0,C 180,E1 -2052.146,E2 -2052.146} C_VEL
LIN {X 0,Y 573.118,Z 243.685,A -85,B 0,C 180,E1 -2054.349,E2 -2054.349} C_VEL
LIN {X 0,Y 573.154,Z 238.739,A -85,B 0,C 180,E1 -2057.249,E2 -2057.249} C_VEL
LIN {X 0,Y 573.235,Z 235.115,A -85,B 0,C 180,E1 -2059.403,E2 -2059.403} C_VEL
LIN {X 0,Y 573.188,Z 232.772,A -85,B 0,C 180,E1 -2060.828,E2 -2060.828} C_VEL
LIN {X 0,Y 573.203,Z 232.084,A -85,B 0,C 180,E1 -2061.54,E2 -2061.54} C_VEL
LIN {X 0,Y 573.233,Z 232.084,A -85,B 0,C 180,E1 -2063.665,E2 -2063.665} C_VEL
LIN {X 0,Y 573.226,Z 232.084,A -85,B 0,C 180,E1 -2065.782,E2 -2065.782} C_VEL
LIN {X 0,Y 573.296,Z 232.073,A -85,B 0,C 180,E1 -2067.893,E2 -2067.893} C_VEL
LIN {X 0,Y 573.328,Z 232.072,A -85,B 0,C 180,E1 -2070.702,E2 -2070.702} C_VEL
LIN {X 0,Y 573.234,Z 232.082,A -85,B 0,C 180,E1 -2073.515,E2 -2073.515} C_VEL
LIN {X 0,Y 573.284,Z 232.078,A -85,B 0,C 180,E1 -2075.628,E2 -2075.628} C_VEL
LIN {X 0,Y 573.3,Z 232.074,A -85,B 0,C 180,E1 -2078.459,E2 -2078.459} C_VEL
LIN {X 0,Y 573.289,Z 232.075,A -85,B 0,C 180,E1 -2081.312,E2 -2081.312} C_VEL
LIN {X 0,Y 573.271,Z 232.077,A -85,B 0,C 180,E1 -2084.425,E2 -2084.425} C_VEL
LIN {X 0,Y 573.251,Z 232.079,A -85,B 0,C 180,E1 -2087.112,E2 -2087.112} C_VEL
LIN {X 0,Y 573.248,Z 232.083,A -85,B 0,C 180,E1 -2090.076,E2 -2090.076} C_VEL
LIN {X 0,Y 573.261,Z 232.078,A -85,B 0,C 180,E1 -2093.154,E2 -2093.154} C_VEL
LIN {X 0,Y 573.278,Z 232.078,A -85,B 0,C 180,E1 -2096.189,E2 -2096.189} C_VEL
LIN {X 0,Y 573.234,Z 232.083,A -85,B 0,C 180,E1 -2098.564,E2 -2098.564} C_VEL
LIN {X 0,Y 573.231,Z 232.084,A -85,B 0,C 180,E1 -2100.992,E2 -2100.992} C_VEL
LIN {X 0,Y 573.25,Z 232.081,A -85,B 0,C 180,E1 -2103.524,E2 -2103.524} C_VEL
LIN {X 0,Y 573.25,Z 232.08,A -85,B 0,C 180,E1 -2106.048,E2 -2106.048} C_VEL
LIN {X 0,Y 573.24,Z 232.08,A -85,B 0,C 180,E1 -2108.701,E2 -2108.701} C_VEL
LIN {X 0,Y 573.243,Z 232.084,A -85,B 0,C 180,E1 -2111.596,E2 -2111.596} C_VEL
LIN {X 0,Y 573.227,Z 232.083,A -85,B 0,C 180,E1 -2114.333,E2 -2114.333} C_VEL
LIN {X 0,Y 573.249,Z 232.081,A -85,B 0,C 180,E1 -2117.357,E2 -2117.357} C_VEL
LIN {X 0,Y 573.238,Z 232.081,A -85,B 0,C 180,E1 -2120.394,E2 -2120.394} C_VEL
LIN {X 0,Y 573.245,Z 232.08,A -85,B 0,C 180,E1 -2123.078,E2 -2123.078} C_VEL
LIN {X 0,Y 573.261,Z 232.079,A -85,B 0,C 180,E1 -2125.672,E2 -2125.672} C_VEL
LIN {X 0,Y 573.241,Z 232.082,A -85,B 0,C 180,E1 -2128.186,E2 -2128.186} C_VEL
LIN {X 0,Y 573.258,Z 232.08,A -85,B 0,C 180,E1 -2130.635,E2 -2130.635} C_VEL
LIN {X 0,Y 573.261,Z 232.079,A -85,B 0,C 180,E1 -2133.501,E2 -2133.501} C_VEL
LIN {X 0,Y 573.225,Z 232.082,A -85,B 0,C 180,E1 -2136.135,E2 -2136.135} C_VEL
LIN {X 0,Y 573.253,Z 232.082,A -85,B 0,C 180,E1 -2139.175,E2 -2139.175} C_VEL
LIN {X 0,Y 573.229,Z 232.084,A -85,B 0,C 180,E1 -2141.413,E2 -2141.413} C_VEL
LIN {X 0,Y 573.25,Z 232.079,A -85,B 0,C 180,E1 -2143.623,E2 -2143.623} C_VEL
LIN {X 0,Y 573.264,Z 232.077,A -85,B 0,C 180,E1 -2145.808,E2 -2145.808} C_VEL
LIN {X 0,Y 573.275,Z 232.079,A -85,B 0,C 180,E1 -2148.735,E2 -2148.735} C_VEL
LIN {X 0,Y 573.301,Z 232.074,A -85,B 0,C 180,E1 -2151.542,E2 -2151.542} C_VEL
LIN {X 0,Y 573.284,Z 232.076,A -85,B 0,C 180,E1 -2154.373,E2 -2154.373} C_VEL
LIN {X 0,Y 573.304,Z 232.073,A -85,B 0,C 180,E1 -2157.893,E2 -2157.893} C_VEL
LIN {X 0,Y 573.33,Z 232.072,A -85,B 0,C 180,E1 -2160.703,E2 -2160.703} C_VEL
LIN {X 0,Y 573.239,Z 232.082,A -85,B 0,C 180,E1 -2163.515,E2 -2163.515} C_VEL
LIN {X 0,Y 573.285,Z 232.078,A -85,B 0,C 180,E1 -2165.629,E2 -2165.629} C_VEL
LIN {X 0,Y 573.279,Z 232.076,A -85,B 0,C 180,E1 -2168.46,E2 -2168.46} C_VEL
LIN {X 0,Y 573.265,Z 232.078,A -85,B 0,C 180,E1 -2171.313,E2 -2171.313} C_VEL
LIN {X 0,Y 573.269,Z 232.079,A -85,B 0,C 180,E1 -2174.194,E2 -2174.194} C_VEL
LIN {X 0,Y 573.254,Z 232.079,A -85,B 0,C 180,E1 -2177.112,E2 -2177.112} C_VEL
LIN {X 0,Y 573.248,Z 232.082,A -85,B 0,C 180,E1 -2180.077,E2 -2180.077} C_VEL
LIN {X 0,Y 573.23,Z 232.082,A -85,B 0,C 180,E1 -2183.1,E2 -2183.1} C_VEL
LIN {X 0,Y 573.25,Z 232.08,A -85,B 0,C 180,E1 -2185.411,E2 -2185.411} C_VEL
LIN {X 0,Y 573.262,Z 232.078,A -85,B 0,C 180,E1 -2188.033,E2 -2188.033} C_VEL
LIN {X 0,Y 573.229,Z 232.085,A -85,B 0,C 180,E1 -2190.884,E2 -2190.884} C_VEL
LIN {X 0,Y 573.237,Z 232.082,A -85,B 0,C 180,E1 -2193.522,E2 -2193.522} C_VEL
LIN {X 0,Y 573.239,Z 232.081,A -85,B 0,C 180,E1 -2196.05,E2 -2196.05} C_VEL
LIN {X 0,Y 573.248,Z 232.08,A -85,B 0,C 180,E1 -2198.702,E2 -2198.702} C_VEL
LIN {X 0,Y 573.228,Z 232.084,A -85,B 0,C 180,E1 -2201.458,E2 -2201.458} C_VEL
LIN {X 0,Y 573.232,Z 232.083,A -85,B 0,C 180,E1 -2204.334,E2 -2204.334} C_VEL
LIN {X 0,Y 573.241,Z 232.082,A -85,B 0,C 180,E1 -2207.359,E2 -2207.359} C_VEL
LIN {X 0,Y 573.247,Z 232.08,A -85,B 0,C 180,E1 -2210.394,E2 -2210.394} C_VEL
LIN {X 0,Y 573.243,Z 232.084,A -85,B 0,C 180,E1 -2213.516,E2 -2213.516} C_VEL
LIN {X 0,Y 573.274,Z 232.323,A -85,B 0,C 180,E1 -2213.736,E2 -2213.736} C_VEL
LIN {X 0,Y 573.578,Z 235.061,A -85,B 0,C 180,E1 -2214.839,E2 -2214.839} C_VEL
LIN {X 0,Y 573.476,Z 242.621,A -85,B 0,C 180,E1 -2217.737,E2 -2217.737} C_VEL
LIN {X 0,Y 573.356,Z 250.072,A -85,B 0,C 180,E1 -2220.494,E2 -2220.494} C_VEL
LIN {X 0,Y 573.271,Z 257.13,A -85,B 0,C 180,E1 -2223.026,E2 -2223.026} C_VEL
LIN {X 0,Y 573.238,Z 265.091,A -85,B 0,C 180,E1 -2225.751,E2 -2225.751} C_VEL
LIN {X 0,Y 573.217,Z 273.899,A -85,B 0,C 180,E1 -2228.719,E2 -2228.719} C_VEL
LIN {X 0,Y 573.16,Z 281.918,A -85,B 0,C 180,E1 -2231.409,E2 -2231.409} C_VEL
LIN {X 0,Y 573.11,Z 290.823,A -85,B 0,C 180,E1 -2234.349,E2 -2234.349} C_VEL
LIN {X 0,Y 573.068,Z 299.727,A -85,B 0,C 180,E1 -2237.247,E2 -2237.247} C_VEL
LIN {X 0,Y 573.049,Z 300.492,A -85,B 0,C 180,E1 -2237.494,E2 -2237.494} C_VEL
LIN {X 0,Y 573.878,Z 306.376,A -85,B 0,C 180,E1 -2237.625,E2 -2237.625} C_VEL
LIN {X 0,Y 573.765,Z 318.504,A -85,B 0,C 180,E1 -2237.937,E2 -2237.937} C_VEL
LIN {X 0,Y 573.65,Z 330.319,A -85,B 0,C 180,E1 -2238.373,E2 -2238.373} C_VEL
LIN {X 0,Y 573.522,Z 342.429,A -85,B 0,C 180,E1 -2238.974,E2 -2238.974} C_VEL
LIN {X 0,Y 573.45,Z 353.483,A -85,B 0,C 180,E1 -2239.675,E2 -2239.675} C_VEL
LIN {X 0,Y 573.308,Z 363.648,A -85,B 0,C 180,E1 -2240.474,E2 -2240.474} C_VEL
LIN {X 0,Y 573.215,Z 372.787,A -85,B 0,C 180,E1 -2241.362,E2 -2241.362} C_VEL
LIN {X 0,Y 573.143,Z 381.69,A -85,B 0,C 180,E1 -2242.425,E2 -2242.425} C_VEL
LIN {X 0,Y 573.051,Z 388.406,A -85,B 0,C 180,E1 -2243.415,E2 -2243.415} C_VEL
LIN {X 0,Y 573.071,Z 393.68,A -85,B 0,C 180,E1 -2244.37,E2 -2244.37} C_VEL
LIN {X 0,Y 573.029,Z 398.372,A -85,B 0,C 180,E1 -2245.427,E2 -2245.427} C_VEL
LIN {X 0,Y 573.022,Z 401.957,A -85,B 0,C 180,E1 -2246.484,E2 -2246.484} C_VEL
LIN {X 0,Y 572.959,Z 403.808,A -85,B 0,C 180,E1 -2247.188,E2 -2247.188} C_VEL
LIN {X 0,Y 572.94,Z 405.198,A -85,B 0,C 180,E1 -2247.891,E2 -2247.891} C_VEL
LIN {X 0,Y 572.941,Z 406.785,A -85,B 0,C 180,E1 -2249.297,E2 -2249.297} C_VEL
LIN {X 0,Y 572.938,Z 407,A -85,B 0,C 180,E1 -2250,E2 -2250} C_VEL
LIN {X 0,Y 572.946,Z 406.186,A -85,B 0,C 180,E1 -2251.406,E2 -2251.406} C_VEL
LIN {X 0,Y 572.94,Z 405.2,A -85,B 0,C 180,E1 -2252.109,E2 -2252.109} C_VEL
LIN {X 0,Y 572.959,Z 403.81,A -85,B 0,C 180,E1 -2252.812,E2 -2252.812} C_VEL
LIN {X 0,Y 573.015,Z 400.896,A -85,B 0,C 180,E1 -2253.868,E2 -2253.868} C_VEL
LIN {X 0,Y 572.963,Z 396.95,A -85,B 0,C 180,E1 -2254.925,E2 -2254.925} C_VEL
LIN {X 0,Y 573.065,Z 390.878,A -85,B 0,C 180,E1 -2256.16,E2 -2256.16} C_VEL
LIN {X 0,Y 573.119,Z 384.239,A -85,B 0,C 180,E1 -2257.221,E2 -2257.221} C_VEL
LIN {X 0,Y 573.201,Z 375.993,A -85,B 0,C 180,E1 -2258.283,E2 -2258.283} C_VEL
LIN {X 0,Y 573.287,Z 367.541,A -85,B 0,C 180,E1 -2259.17,E2 -2259.17} C_VEL
LIN {X 0,Y 573.43,Z 357.102,A -85,B 0,C 180,E1 -2260.058,E2 -2260.058} C_VEL
LIN {X 0,Y 573.512,Z 345.537,A -85,B 0,C 180,E1 -2260.847,E2 -2260.847} C_VEL
LIN {X 0,Y 573.61,Z 333.891,A -85,B 0,C 180,E1 -2261.466,E2 -2261.466} C_VEL
LIN {X 0,Y 573.748,Z 321.181,A -85,B 0,C 180,E1 -2261.974,E2 -2261.974} C_VEL
LIN {X 0,Y 573.856,Z 308.533,A -85,B 0,C 180,E1 -2262.331,E2 -2262.331} C_VEL
LIN {X 0,Y 573.683,Z 304.546,A -85,B 0,C 180,E1 -2262.415,E2 -2262.415} C_VEL
LIN {X 0,Y 573.049,Z 300.493,A -85,B 0,C 180,E1 -2262.506,E2 -2262.506} C_VEL
LIN {X 0,Y 573.086,Z 291.936,A -85,B 0,C 180,E1 -2265.287,E2 -2265.287} C_VEL
LIN {X 0,Y 573.149,Z 284.145,A -85,B 0,C 180,E1 -2267.851,E2 -2267.851} C_VEL
LIN {X 0,Y 573.193,Z 276.354,A -85,B 0,C 180,E1 -2270.453,E2 -2270.453} C_VEL
LIN {X 0,Y 573.213,Z 268.345,A -85,B 0,C 180,E1 -2273.138,E2 -2273.138} C_VEL
LIN {X 0,Y 573.253,Z 260.41,A -85,B 0,C 180,E1 -2275.799,E2 -2275.799} C_VEL
LIN {X 0,Y 573.311,Z 252.615,A -85,B 0,C 180,E1 -2278.56,E2 -2278.56} C_VEL
LIN {X 0,Y 573.426,Z 244.865,A -85,B 0,C 180,E1 -2281.391,E2 -2281.391} C_VEL
LIN {X 0,Y 573.521,Z 239.111,A -85,B 0,C 180,E1 -2283.562,E2 -2283.562} C_VEL
LIN {X 0,Y 573.559,Z 233.977,A -85,B 0,C 180,E1 -2285.581,E2 -2285.581} C_VEL
LIN {X 0,Y 573.304,Z 232.076,A -85,B 0,C 180,E1 -2286.371,E2 -2286.371} C_VEL
LIN {X 0,Y 573.238,Z 232.083,A -85,B 0,C 180,E1 -2289.607,E2 -2289.607} C_VEL
LIN {X 0,Y 573.243,Z 232.082,A -85,B 0,C 180,E1 -2292.641,E2 -2292.641} C_VEL
LIN {X 0,Y 573.233,Z 232.084,A -85,B 0,C 180,E1 -2295.666,E2 -2295.666} C_VEL
LIN {X 0,Y 573.243,Z 232.084,A -85,B 0,C 180,E1 -2298.543,E2 -2298.543} C_VEL
LIN {X 0,Y 573.246,Z 232.082,A -85,B 0,C 180,E1 -2301.298,E2 -2301.298} C_VEL
LIN {X 0,Y 573.261,Z 232.079,A -85,B 0,C 180,E1 -2304.01,E2 -2304.01} C_VEL
LIN {X 0,Y 573.281,Z 232.077,A -85,B 0,C 180,E1 -2306.518,E2 -2306.518} C_VEL
LIN {X 0,Y 573.241,Z 232.082,A -85,B 0,C 180,E1 -2309.114,E2 -2309.114} C_VEL
LIN {X 0,Y 573.259,Z 232.081,A -85,B 0,C 180,E1 -2311.967,E2 -2311.967} C_VEL
LIN {X 0,Y 573.249,Z 232.081,A -85,B 0,C 180,E1 -2314.589,E2 -2314.589} C_VEL
LIN {X 0,Y 573.232,Z 232.083,A -85,B 0,C 180,E1 -2317.661,E2 -2317.661} C_VEL
LIN {X 0,Y 573.271,Z 232.078,A -85,B 0,C 180,E1 -2320.727,E2 -2320.727} C_VEL
LIN {X 0,Y 573.253,Z 232.08,A -85,B 0,C 180,E1 -2323.621,E2 -2323.621} C_VEL
LIN {X 0,Y 573.234,Z 232.083,A -85,B 0,C 180,E1 -2326.529,E2 -2326.529} C_VEL
LIN {X 0,Y 573.276,Z 232.077,A -85,B 0,C 180,E1 -2328.733,E2 -2328.733} C_VEL
LIN {X 0,Y 573.302,Z 232.075,A -85,B 0,C 180,E1 -2331.54,E2 -2331.54} C_VEL
LIN {X 0,Y 573.287,Z 232.078,A -85,B 0,C 180,E1 -2334.371,E2 -2334.371} C_VEL
LIN {X 0,Y 573.3,Z 232.074,A -85,B 0,C 180,E1 -2337.892,E2 -2337.892} C_VEL
